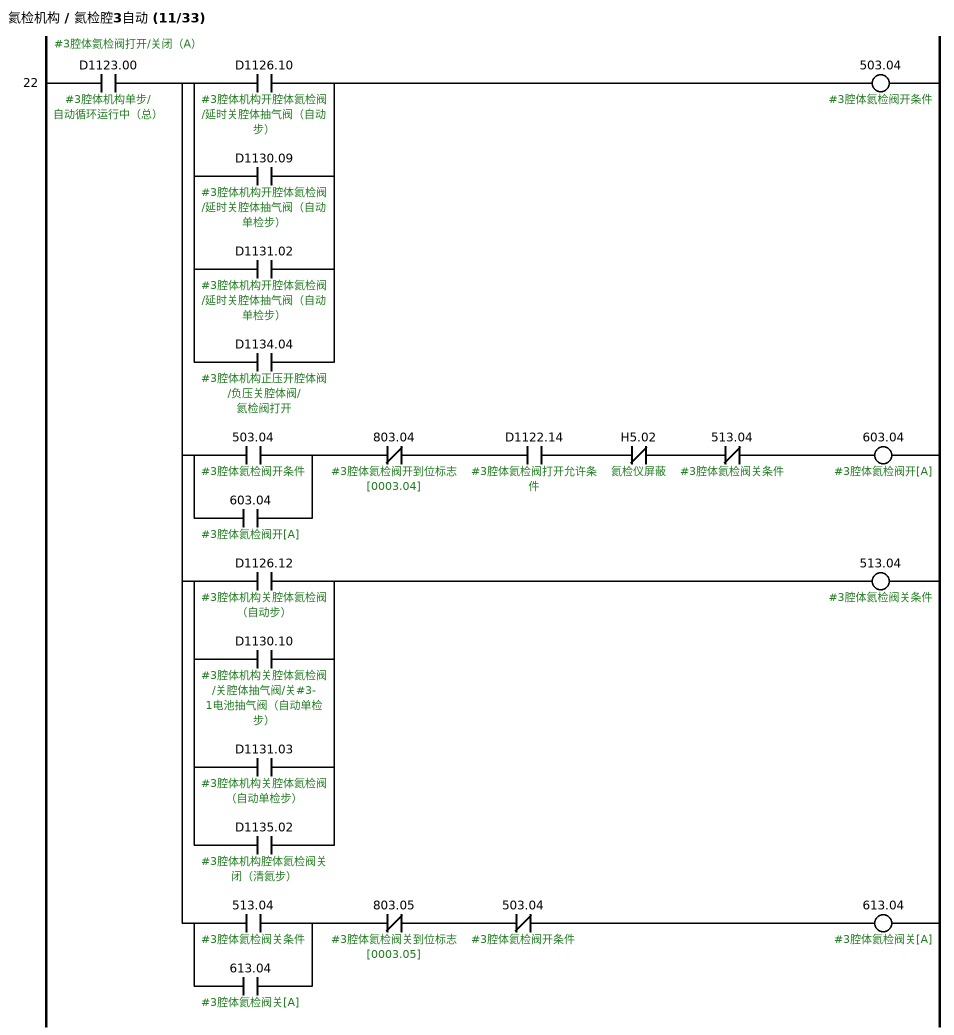
; [picture p312: 氦检机构 / 氦检腔3自动, rungs 22-22]
; rung 22: #3腔体氦检阀打开/关闭（A）
LD D1123.00  ; #3腔体机构单步/自动循环运行中（总）
OUT TR0
LD D1126.10  ; #3腔体机构开腔体氦检阀/延时关腔体抽气阀（自动步）
OR D1130.09  ; #3腔体机构开腔体氦检阀/延时关腔体抽气阀（自动单检步）
OR D1131.02  ; #3腔体机构开腔体氦检阀/延时关腔体抽气阀（自动单检步）
OR D1134.04  ; #3腔体机构正压开腔体阀/负压关腔体阀/氦检阀打开
ANDLD
OUT 503.04  ; #3腔体氦检阀开条件
LD TR0
LD 503.04  ; #3腔体氦检阀开条件
OR 603.04  ; #3腔体氦检阀开[A]
ANDLD
ANDNOT 803.04  ; #3腔体氦检阀开到位标志[0003.04]
AND D1122.14  ; #3腔体氦检阀打开允许条件
ANDNOT H5.02  ; 氦检仪屏蔽
ANDNOT 513.04  ; #3腔体氦检阀关条件
OUT 603.04  ; #3腔体氦检阀开[A]
LD TR0
LD D1126.12  ; #3腔体机构关腔体氦检阀（自动步）
OR D1130.10  ; #3腔体机构关腔体氦检阀/关腔体抽气阀/关#3-1电池抽气阀（自动单检步）
OR D1131.03  ; #3腔体机构关腔体氦检阀（自动单检步）
OR D1135.02  ; #3腔体机构腔体氦检阀关闭（清氦步）
ANDLD
OUT 513.04  ; #3腔体氦检阀关条件
LD TR0
LD 513.04  ; #3腔体氦检阀关条件
OR 613.04  ; #3腔体氦检阀关[A]
ANDLD
ANDNOT 803.05  ; #3腔体氦检阀关到位标志[0003.05]
ANDNOT 503.04  ; #3腔体氦检阀开条件
OUT 613.04  ; #3腔体氦检阀关[A]

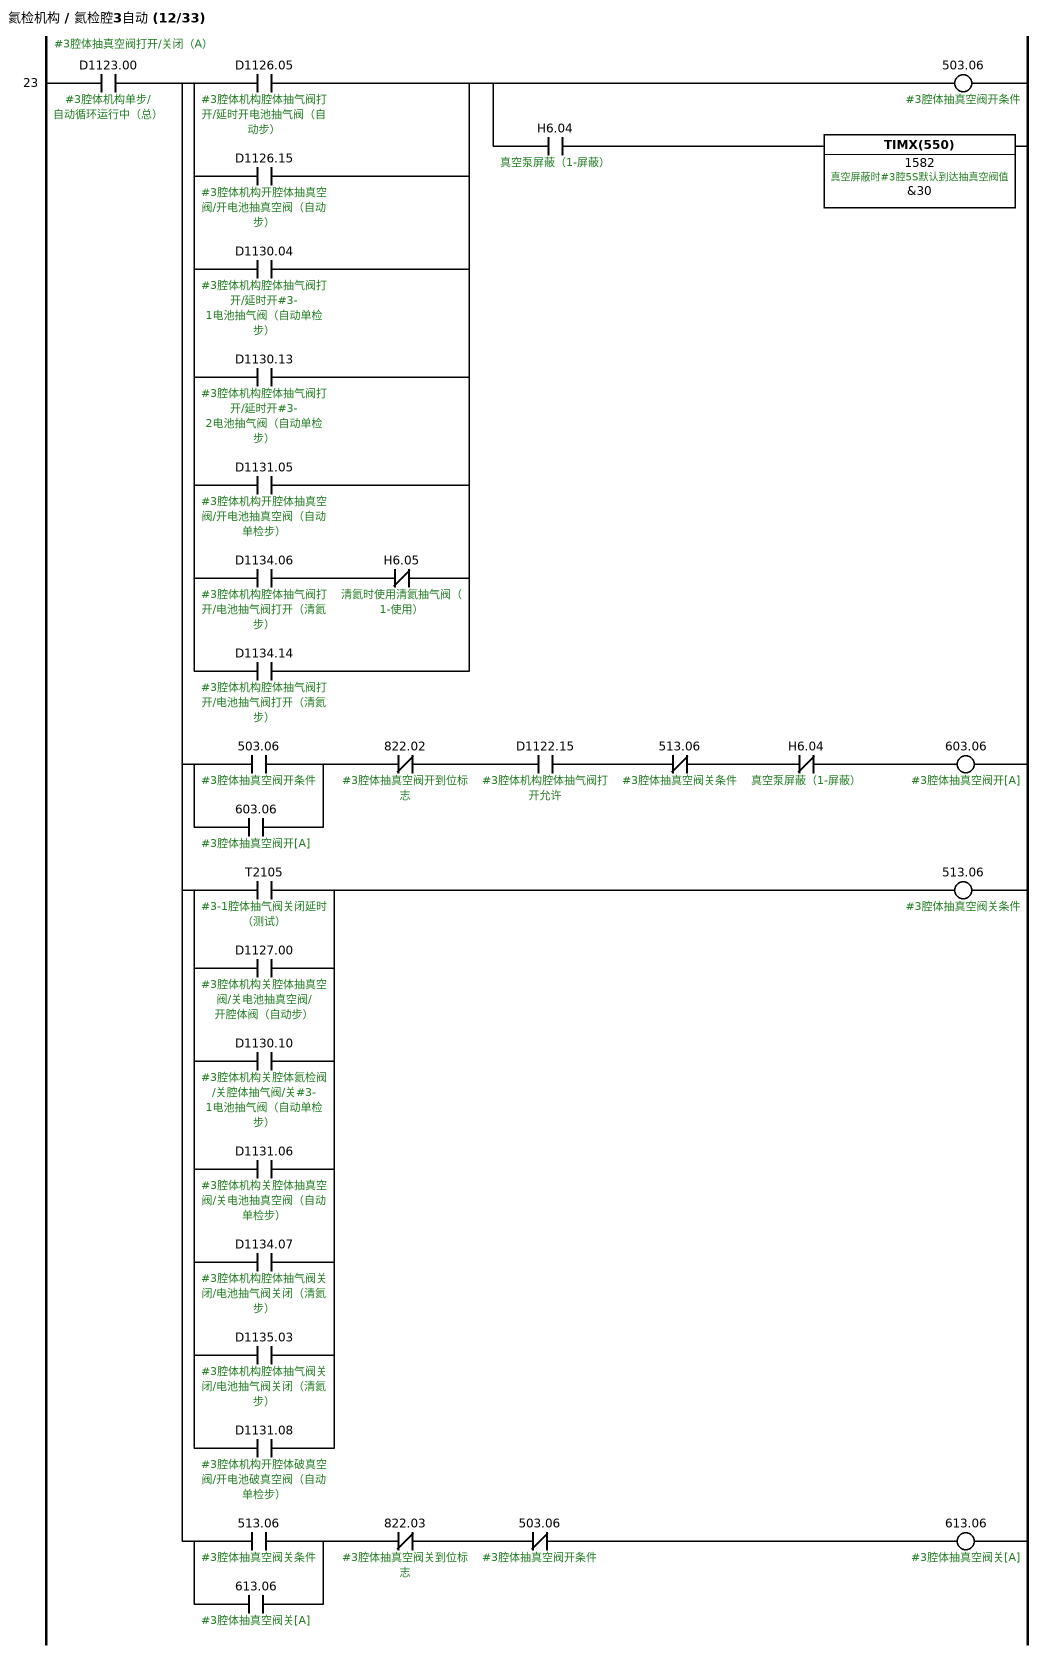
; rung 23: #3腔体抽真空阀打开/关闭（A）
LD D1123.00  ; #3腔体机构单步/自动循环运行中（总）
OUT TR0
LD D1126.05  ; #3腔体机构腔体抽气阀打开/延时开电池抽气阀（自动步）
OR D1126.15  ; #3腔体机构开腔体抽真空阀/开电池抽真空阀（自动步）
OR D1130.04  ; #3腔体机构腔体抽气阀打开/延时开#3-1电池抽气阀（自动单检步）
OR D1130.13  ; #3腔体机构腔体抽气阀打开/延时开#3-2电池抽气阀（自动单检步）
OR D1131.05  ; #3腔体机构开腔体抽真空阀/开电池抽真空阀（自动单检步）
LD D1134.06  ; #3腔体机构腔体抽气阀打开/电池抽气阀打开（清氦步）
ANDNOT H6.05  ; 清氦时使用清氦抽气阀（1-使用）
ORLD
OR D1134.14  ; #3腔体机构腔体抽气阀打开/电池抽气阀打开（清氦步）
ANDLD
OUT 503.06  ; #3腔体抽真空阀开条件
AND H6.04  ; 真空泵屏蔽（1-屏蔽）
TIMX(550) 1582 &30  ; 真空屏蔽时#3腔5S默认到达抽真空阀值
LD TR0
LD 503.06  ; #3腔体抽真空阀开条件
OR 603.06  ; #3腔体抽真空阀开[A]
ANDLD
ANDNOT 822.02  ; #3腔体抽真空阀开到位标志
AND D1122.15  ; #3腔体机构腔体抽气阀打开允许
ANDNOT 513.06  ; #3腔体抽真空阀关条件
ANDNOT H6.04  ; 真空泵屏蔽（1-屏蔽）
OUT 603.06  ; #3腔体抽真空阀开[A]
LD TR0
LD T2105  ; #3-1腔体抽气阀关闭延时（测试）
OR D1127.00  ; #3腔体机构关腔体抽真空阀/关电池抽真空阀/开腔体阀（自动步）
OR D1130.10  ; #3腔体机构关腔体氦检阀/关腔体抽气阀/关#3-1电池抽气阀（自动单检步）
OR D1131.06  ; #3腔体机构关腔体抽真空阀/关电池抽真空阀（自动单检步）
OR D1134.07  ; #3腔体机构腔体抽气阀关闭/电池抽气阀关闭（清氦步）
OR D1135.03  ; #3腔体机构腔体抽气阀关闭/电池抽气阀关闭（清氦步）
OR D1131.08  ; #3腔体机构开腔体破真空阀/开电池破真空阀（自动单检步）
ANDLD
OUT 513.06  ; #3腔体抽真空阀关条件
LD TR0
LD 513.06  ; #3腔体抽真空阀关条件
OR 613.06  ; #3腔体抽真空阀关[A]
ANDLD
ANDNOT 822.03  ; #3腔体抽真空阀关到位标志
ANDNOT 503.06  ; #3腔体抽真空阀开条件
OUT 613.06  ; #3腔体抽真空阀关[A]

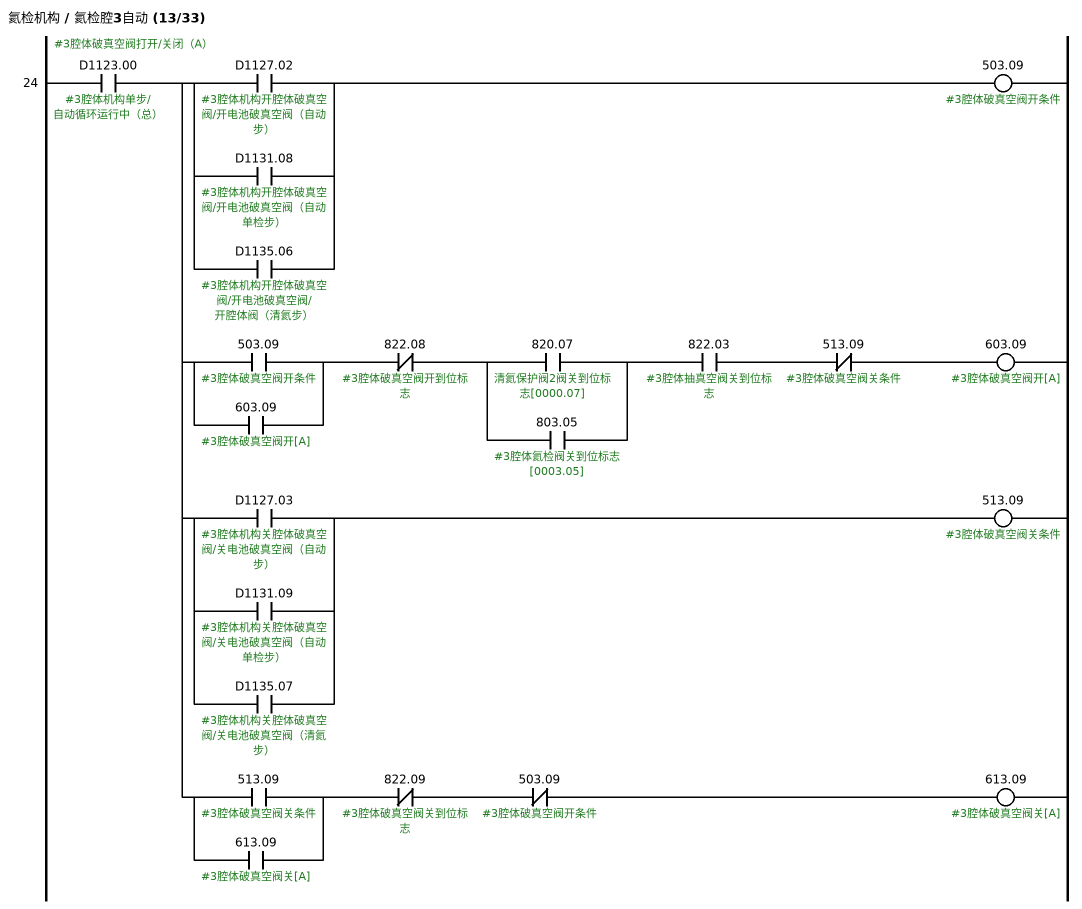
; rung 24: #3腔体破真空阀打开/关闭（A）
LD D1123.00  ; #3腔体机构单步/自动循环运行中（总）
OUT TR0
LD D1127.02  ; #3腔体机构开腔体破真空阀/开电池破真空阀（自动步）
OR D1131.08  ; #3腔体机构开腔体破真空阀/开电池破真空阀（自动单检步）
OR D1135.06  ; #3腔体机构开腔体破真空阀/开电池破真空阀/开腔体阀（清氦步）
ANDLD
OUT 503.09  ; #3腔体破真空阀开条件
LD TR0
LD 503.09  ; #3腔体破真空阀开条件
OR 603.09  ; #3腔体破真空阀开[A]
ANDLD
ANDNOT 822.08  ; #3腔体破真空阀开到位标志
LD 820.07  ; 清氦保护阀2阀关到位标志[0000.07]
OR 803.05  ; #3腔体氦检阀关到位标志[0003.05]
ANDLD
AND 822.03  ; #3腔体抽真空阀关到位标志
ANDNOT 513.09  ; #3腔体破真空阀关条件
OUT 603.09  ; #3腔体破真空阀开[A]
LD TR0
LD D1127.03  ; #3腔体机构关腔体破真空阀/关电池破真空阀（自动步）
OR D1131.09  ; #3腔体机构关腔体破真空阀/关电池破真空阀（自动单检步）
OR D1135.07  ; #3腔体机构关腔体破真空阀/关电池破真空阀（清氦步）
ANDLD
OUT 513.09  ; #3腔体破真空阀关条件
LD TR0
LD 513.09  ; #3腔体破真空阀关条件
OR 613.09  ; #3腔体破真空阀关[A]
ANDLD
ANDNOT 822.09  ; #3腔体破真空阀关到位标志
ANDNOT 503.09  ; #3腔体破真空阀开条件
OUT 613.09  ; #3腔体破真空阀关[A]

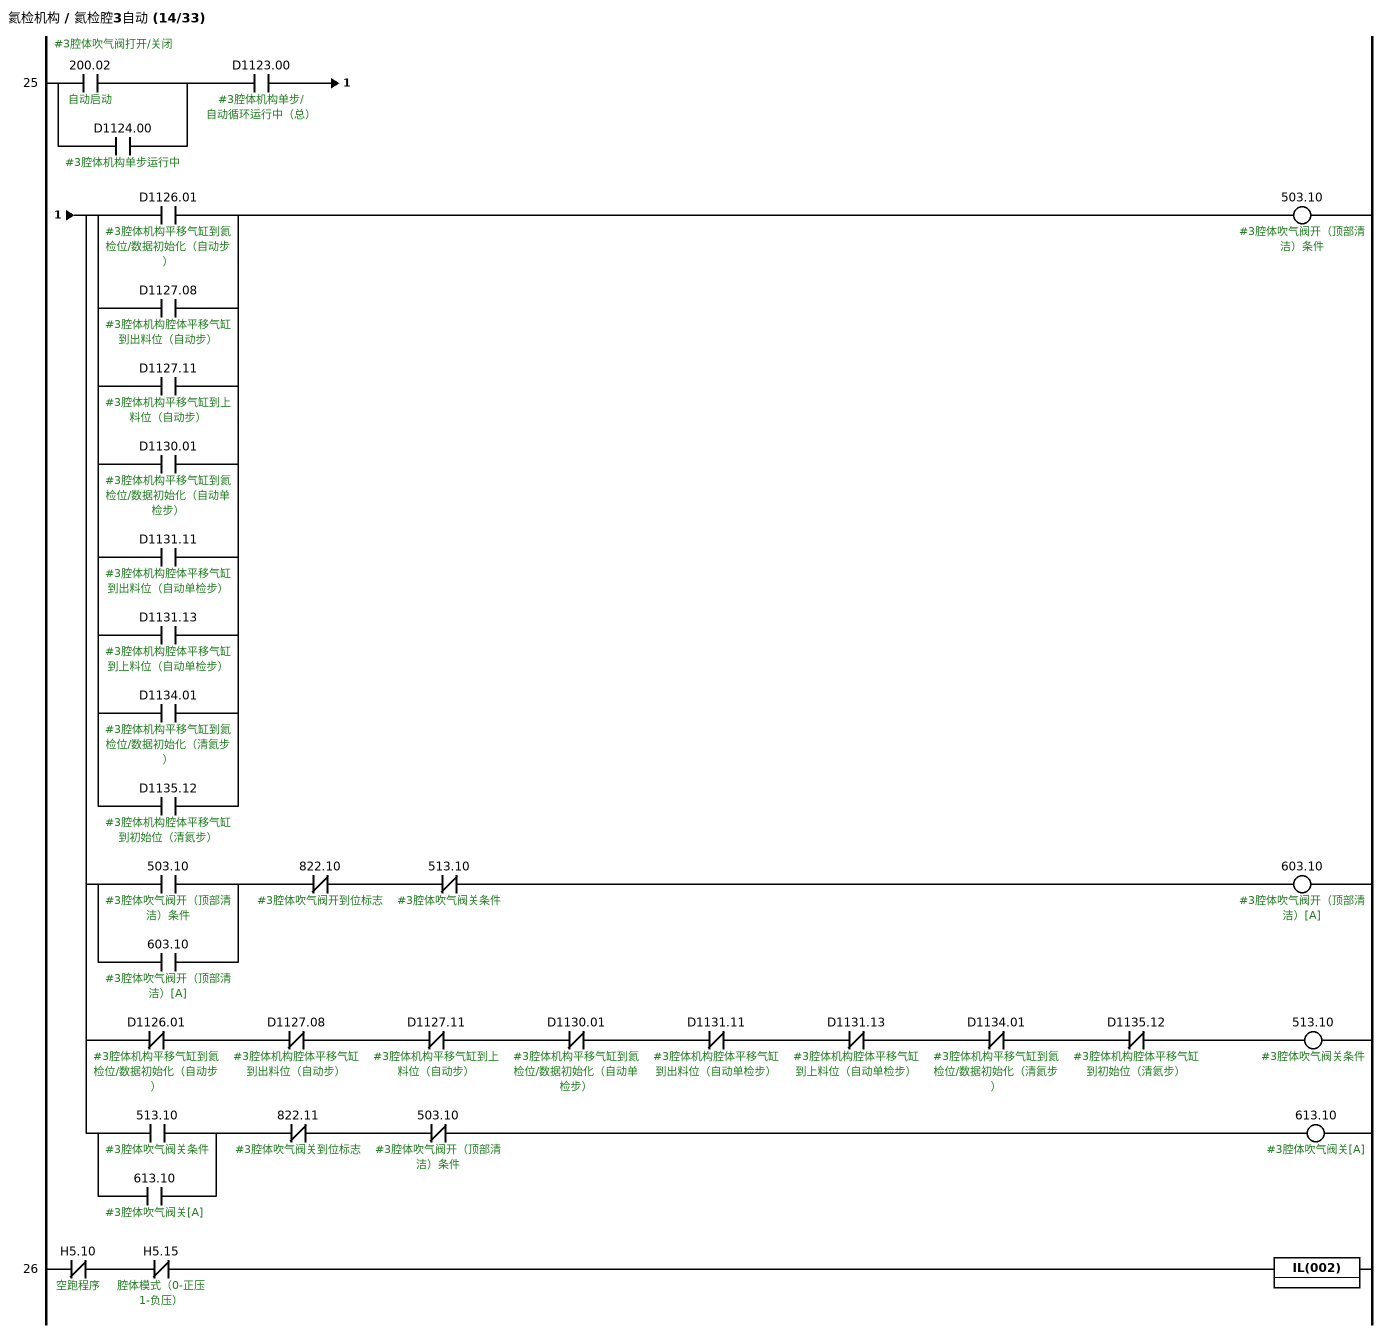
; rung 25: #3腔体吹气阀打开/关闭
LD 200.02  ; 自动启动
OR D1124.00  ; #3腔体机构单步运行中
AND D1123.00  ; #3腔体机构单步/自动循环运行中（总）
OUT TR0
LD D1126.01  ; #3腔体机构平移气缸到氦检位/数据初始化（自动步）
OR D1127.08  ; #3腔体机构腔体平移气缸到出料位（自动步）
OR D1127.11  ; #3腔体机构平移气缸到上料位（自动步）
OR D1130.01  ; #3腔体机构平移气缸到氦检位/数据初始化（自动单检步）
OR D1131.11  ; #3腔体机构腔体平移气缸到出料位（自动单检步）
OR D1131.13  ; #3腔体机构腔体平移气缸到上料位（自动单检步）
OR D1134.01  ; #3腔体机构平移气缸到氦检位/数据初始化（清氦步）
OR D1135.12  ; #3腔体机构腔体平移气缸到初始位（清氦步）
ANDLD
OUT 503.10  ; #3腔体吹气阀开（顶部清洁）条件
LD TR0
LD 503.10  ; #3腔体吹气阀开（顶部清洁）条件
OR 603.10  ; #3腔体吹气阀开（顶部清洁）[A]
ANDLD
ANDNOT 822.10  ; #3腔体吹气阀开到位标志
ANDNOT 513.10  ; #3腔体吹气阀关条件
OUT 603.10  ; #3腔体吹气阀开（顶部清洁）[A]
LD TR0
ANDNOT D1126.01  ; #3腔体机构平移气缸到氦检位/数据初始化（自动步）
ANDNOT D1127.08  ; #3腔体机构腔体平移气缸到出料位（自动步）
ANDNOT D1127.11  ; #3腔体机构平移气缸到上料位（自动步）
ANDNOT D1130.01  ; #3腔体机构平移气缸到氦检位/数据初始化（自动单检步）
ANDNOT D1131.11  ; #3腔体机构腔体平移气缸到出料位（自动单检步）
ANDNOT D1131.13  ; #3腔体机构腔体平移气缸到上料位（自动单检步）
ANDNOT D1134.01  ; #3腔体机构平移气缸到氦检位/数据初始化（清氦步）
ANDNOT D1135.12  ; #3腔体机构腔体平移气缸到初始位（清氦步）
OUT 513.10  ; #3腔体吹气阀关条件
LD TR0
LD 513.10  ; #3腔体吹气阀关条件
OR 613.10  ; #3腔体吹气阀关[A]
ANDLD
ANDNOT 822.11  ; #3腔体吹气阀关到位标志
ANDNOT 503.10  ; #3腔体吹气阀开（顶部清洁）条件
OUT 613.10  ; #3腔体吹气阀关[A]
; rung 26
LDNOT H5.10  ; 空跑程序
ANDNOT H5.15  ; 腔体模式（0-正压 1-负压）
IL(002)

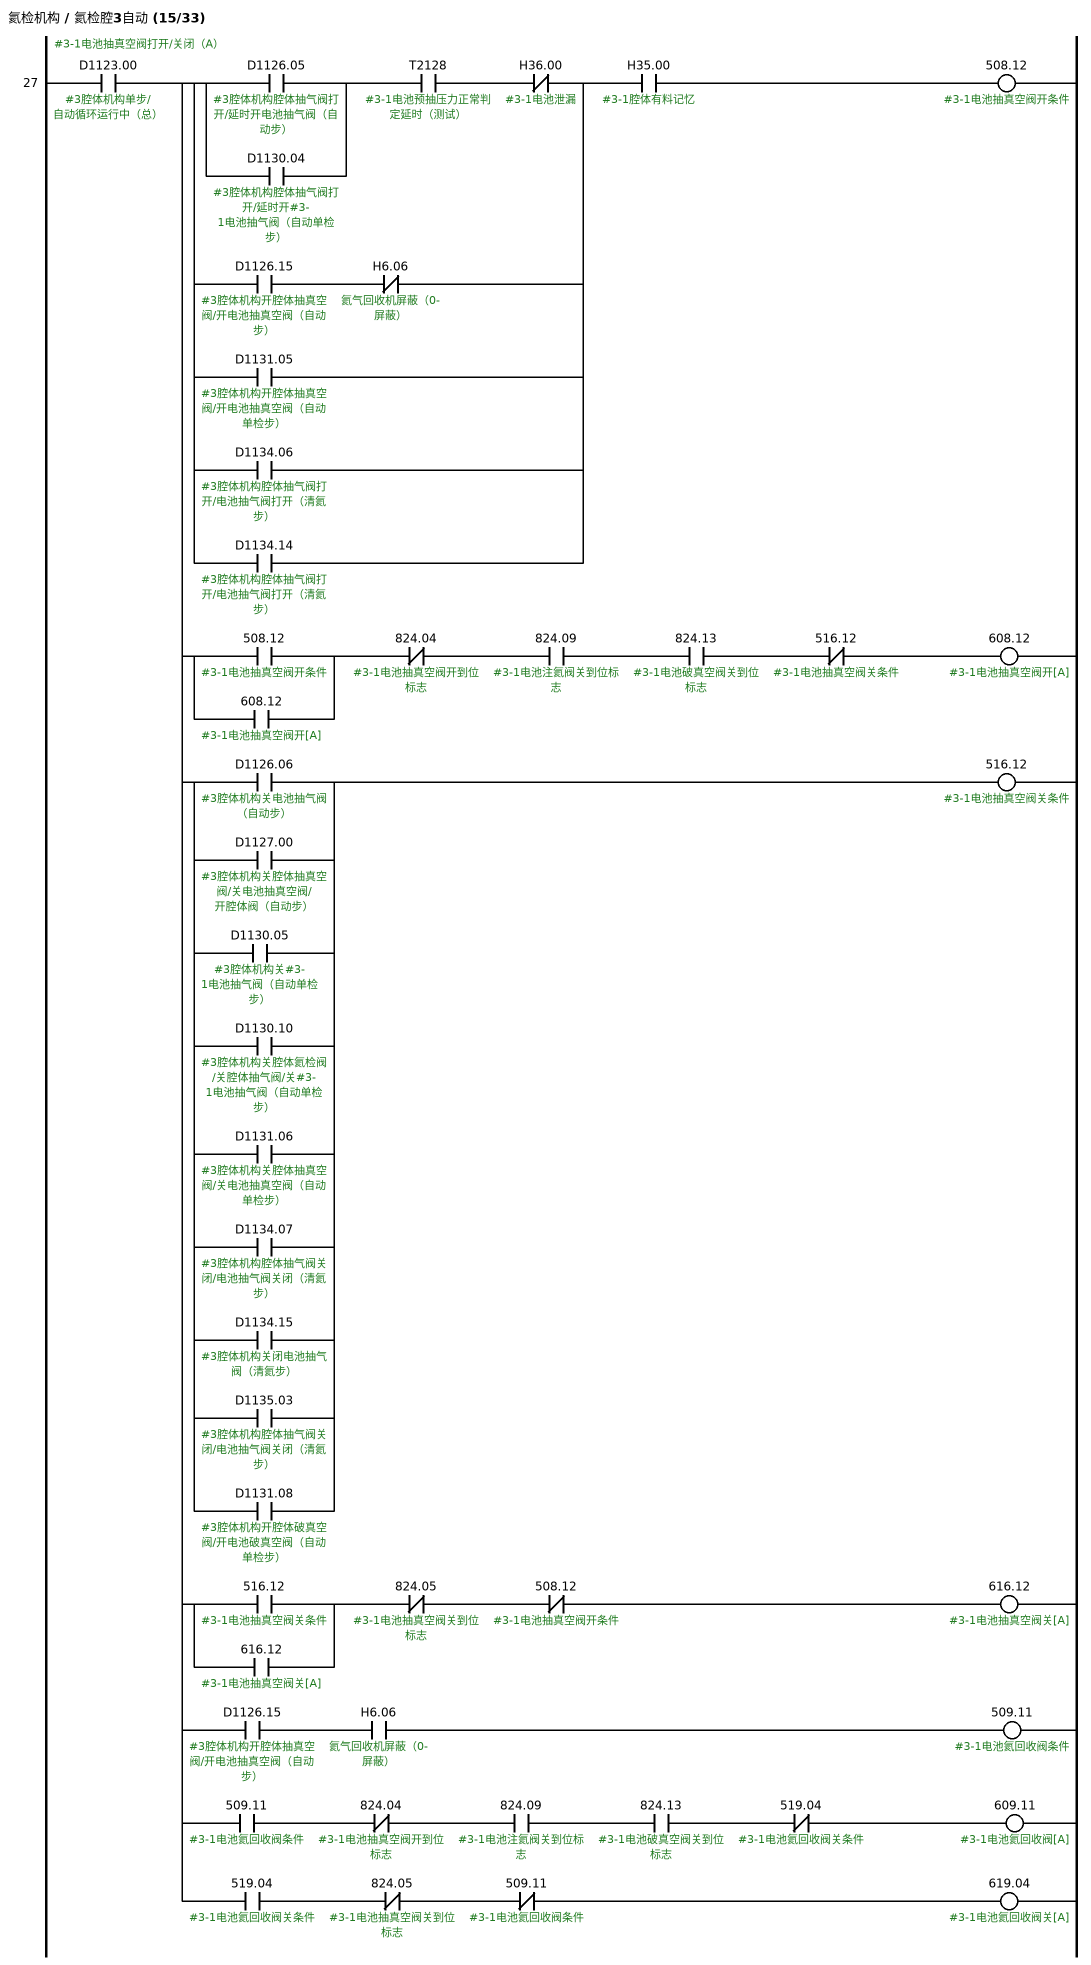
; rung 27: #3-1电池抽真空阀打开/关闭（A）
LD D1123.00  ; #3腔体机构单步/自动循环运行中（总）
OUT TR0
LD D1126.05  ; #3腔体机构腔体抽气阀打开/延时开电池抽气阀（自动步）
OR D1130.04  ; #3腔体机构腔体抽气阀打开/延时开#3-1电池抽气阀（自动单检步）
AND T2128  ; #3-1电池预抽压力正常判定延时（测试）
ANDNOT H36.00  ; #3-1电池泄漏
LD D1126.15  ; #3腔体机构开腔体抽真空阀/开电池抽真空阀（自动步）
ANDNOT H6.06  ; 氦气回收机屏蔽（0-屏蔽）
ORLD
OR D1131.05  ; #3腔体机构开腔体抽真空阀/开电池抽真空阀（自动单检步）
OR D1134.06  ; #3腔体机构腔体抽气阀打开/电池抽气阀打开（清氦步）
OR D1134.14  ; #3腔体机构腔体抽气阀打开/电池抽气阀打开（清氦步）
ANDLD
AND H35.00  ; #3-1腔体有料记忆
OUT 508.12  ; #3-1电池抽真空阀开条件
LD TR0
LD 508.12  ; #3-1电池抽真空阀开条件
OR 608.12  ; #3-1电池抽真空阀开[A]
ANDLD
ANDNOT 824.04  ; #3-1电池抽真空阀开到位标志
AND 824.09  ; #3-1电池注氦阀关到位标志
AND 824.13  ; #3-1电池破真空阀关到位标志
ANDNOT 516.12  ; #3-1电池抽真空阀关条件
OUT 608.12  ; #3-1电池抽真空阀开[A]
LD TR0
LD D1126.06  ; #3腔体机构关电池抽气阀（自动步）
OR D1127.00  ; #3腔体机构关腔体抽真空阀/关电池抽真空阀/开腔体阀（自动步）
OR D1130.05  ; #3腔体机构关#3-1电池抽气阀（自动单检步）
OR D1130.10  ; #3腔体机构关腔体氦检阀/关腔体抽气阀/关#3-1电池抽气阀（自动单检步）
OR D1131.06  ; #3腔体机构关腔体抽真空阀/关电池抽真空阀（自动单检步）
OR D1134.07  ; #3腔体机构腔体抽气阀关闭/电池抽气阀关闭（清氦步）
OR D1134.15  ; #3腔体机构关闭电池抽气阀（清氦步）
OR D1135.03  ; #3腔体机构腔体抽气阀关闭/电池抽气阀关闭（清氦步）
OR D1131.08  ; #3腔体机构开腔体破真空阀/开电池破真空阀（自动单检步）
ANDLD
OUT 516.12  ; #3-1电池抽真空阀关条件
LD TR0
LD 516.12  ; #3-1电池抽真空阀关条件
OR 616.12  ; #3-1电池抽真空阀关[A]
ANDLD
ANDNOT 824.05  ; #3-1电池抽真空阀关到位标志
ANDNOT 508.12  ; #3-1电池抽真空阀开条件
OUT 616.12  ; #3-1电池抽真空阀关[A]
LD TR0
AND D1126.15  ; #3腔体机构开腔体抽真空阀/开电池抽真空阀（自动步）
AND H6.06  ; 氦气回收机屏蔽（0-屏蔽）
OUT 509.11  ; #3-1电池氦回收阀条件
LD TR0
AND 509.11  ; #3-1电池氦回收阀条件
ANDNOT 824.04  ; #3-1电池抽真空阀开到位标志
AND 824.09  ; #3-1电池注氦阀关到位标志
AND 824.13  ; #3-1电池破真空阀关到位标志
ANDNOT 519.04  ; #3-1电池氦回收阀关条件
OUT 609.11  ; #3-1电池氦回收阀[A]
LD TR0
AND 519.04  ; #3-1电池氦回收阀关条件
ANDNOT 824.05  ; #3-1电池抽真空阀关到位标志
ANDNOT 509.11  ; #3-1电池氦回收阀条件
OUT 619.04  ; #3-1电池氦回收阀关[A]

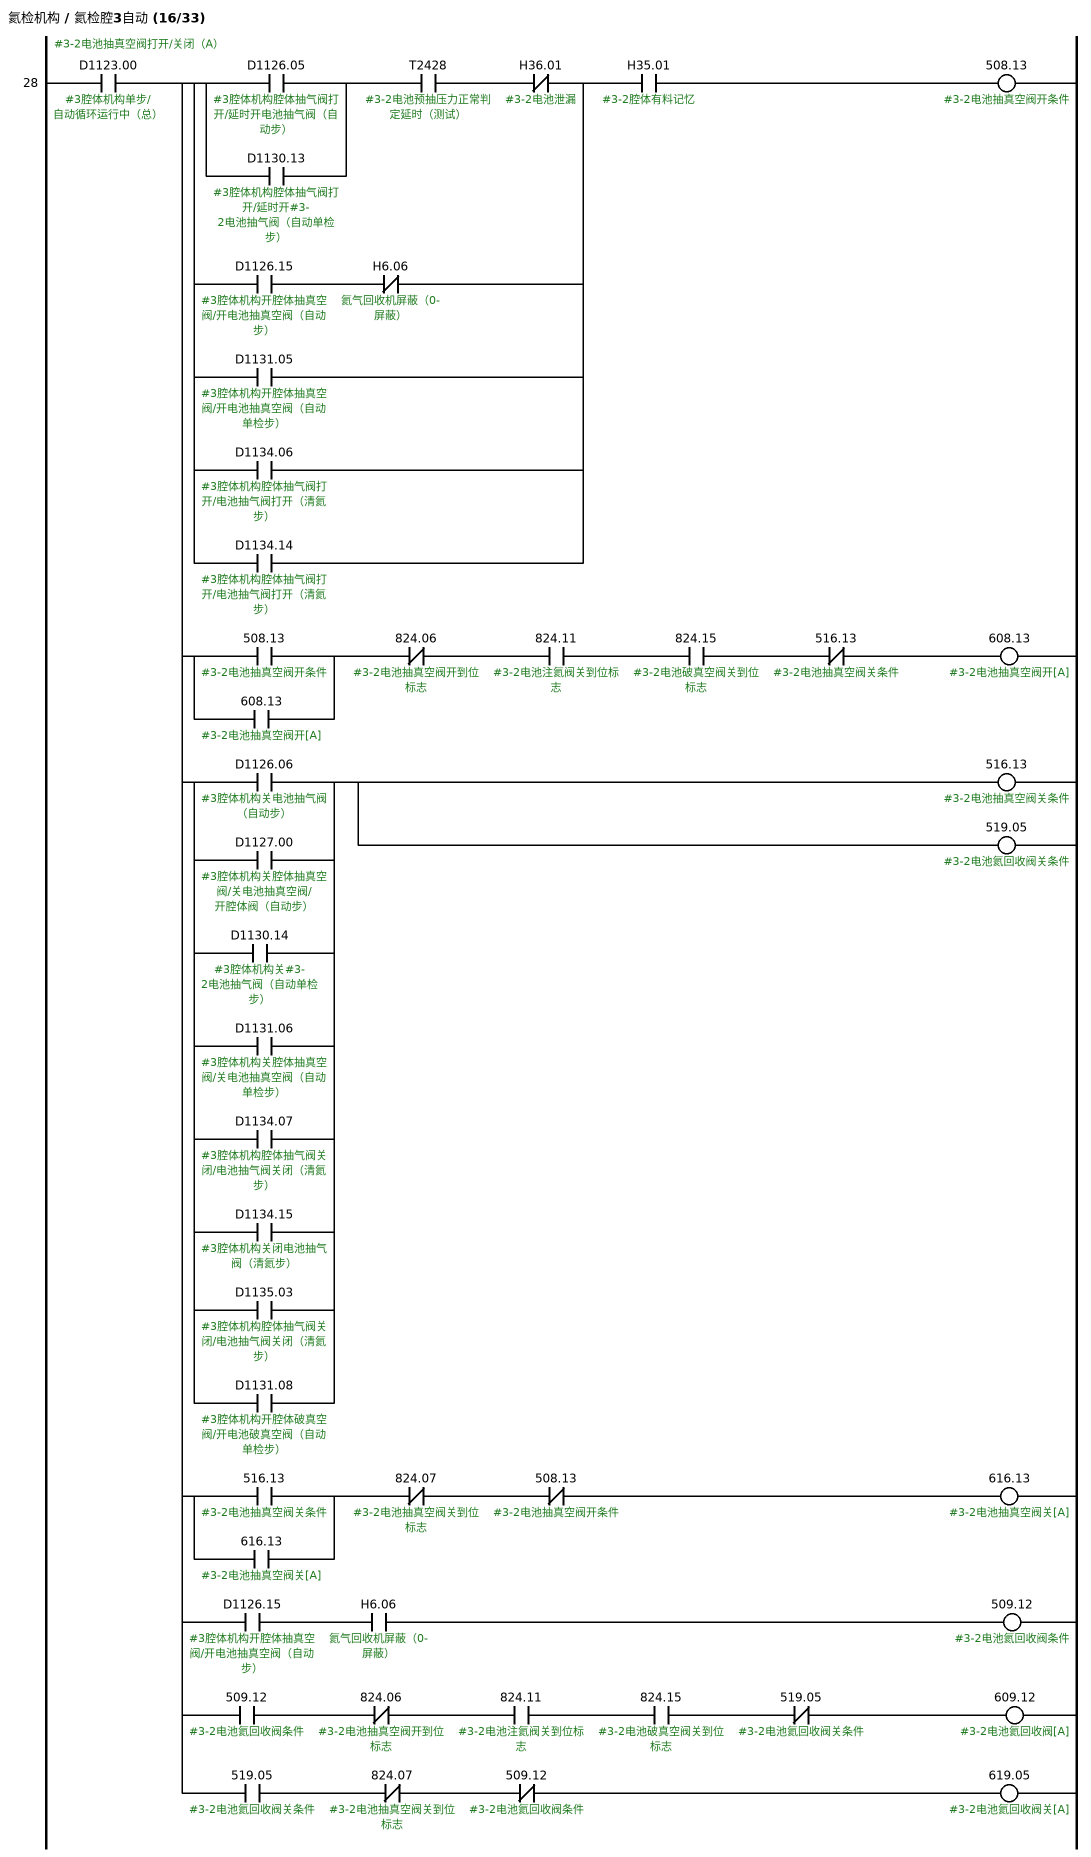
; rung 28: #3-2电池抽真空阀打开/关闭（A）
LD D1123.00  ; #3腔体机构单步/自动循环运行中（总）
OUT TR0
LD D1126.05  ; #3腔体机构腔体抽气阀打开/延时开电池抽气阀（自动步）
OR D1130.13  ; #3腔体机构腔体抽气阀打开/延时开#3-2电池抽气阀（自动单检步）
AND T2428  ; #3-2电池预抽压力正常判定延时（测试）
ANDNOT H36.01  ; #3-2电池泄漏
LD D1126.15  ; #3腔体机构开腔体抽真空阀/开电池抽真空阀（自动步）
ANDNOT H6.06  ; 氦气回收机屏蔽（0-屏蔽）
ORLD
OR D1131.05  ; #3腔体机构开腔体抽真空阀/开电池抽真空阀（自动单检步）
OR D1134.06  ; #3腔体机构腔体抽气阀打开/电池抽气阀打开（清氦步）
OR D1134.14  ; #3腔体机构腔体抽气阀打开/电池抽气阀打开（清氦步）
ANDLD
AND H35.01  ; #3-2腔体有料记忆
OUT 508.13  ; #3-2电池抽真空阀开条件
LD TR0
LD 508.13  ; #3-2电池抽真空阀开条件
OR 608.13  ; #3-2电池抽真空阀开[A]
ANDLD
ANDNOT 824.06  ; #3-2电池抽真空阀开到位标志
AND 824.11  ; #3-2电池注氦阀关到位标志
AND 824.15  ; #3-2电池破真空阀关到位标志
ANDNOT 516.13  ; #3-2电池抽真空阀关条件
OUT 608.13  ; #3-2电池抽真空阀开[A]
LD TR0
LD D1126.06  ; #3腔体机构关电池抽气阀（自动步）
OR D1127.00  ; #3腔体机构关腔体抽真空阀/关电池抽真空阀/开腔体阀（自动步）
OR D1130.14  ; #3腔体机构关#3-2电池抽气阀（自动单检步）
OR D1131.06  ; #3腔体机构关腔体抽真空阀/关电池抽真空阀（自动单检步）
OR D1134.07  ; #3腔体机构腔体抽气阀关闭/电池抽气阀关闭（清氦步）
OR D1134.15  ; #3腔体机构关闭电池抽气阀（清氦步）
OR D1135.03  ; #3腔体机构腔体抽气阀关闭/电池抽气阀关闭（清氦步）
OR D1131.08  ; #3腔体机构开腔体破真空阀/开电池破真空阀（自动单检步）
ANDLD
OUT 516.13  ; #3-2电池抽真空阀关条件
OUT 519.05  ; #3-2电池氦回收阀关条件
LD TR0
LD 516.13  ; #3-2电池抽真空阀关条件
OR 616.13  ; #3-2电池抽真空阀关[A]
ANDLD
ANDNOT 824.07  ; #3-2电池抽真空阀关到位标志
ANDNOT 508.13  ; #3-2电池抽真空阀开条件
OUT 616.13  ; #3-2电池抽真空阀关[A]
LD TR0
AND D1126.15  ; #3腔体机构开腔体抽真空阀/开电池抽真空阀（自动步）
AND H6.06  ; 氦气回收机屏蔽（0-屏蔽）
OUT 509.12  ; #3-2电池氦回收阀条件
LD TR0
AND 509.12  ; #3-2电池氦回收阀条件
ANDNOT 824.06  ; #3-2电池抽真空阀开到位标志
AND 824.11  ; #3-2电池注氦阀关到位标志
AND 824.15  ; #3-2电池破真空阀关到位标志
ANDNOT 519.05  ; #3-2电池氦回收阀关条件
OUT 609.12  ; #3-2电池氦回收阀[A]
LD TR0
AND 519.05  ; #3-2电池氦回收阀关条件
ANDNOT 824.07  ; #3-2电池抽真空阀关到位标志
ANDNOT 509.12  ; #3-2电池氦回收阀条件
OUT 619.05  ; #3-2电池氦回收阀关[A]

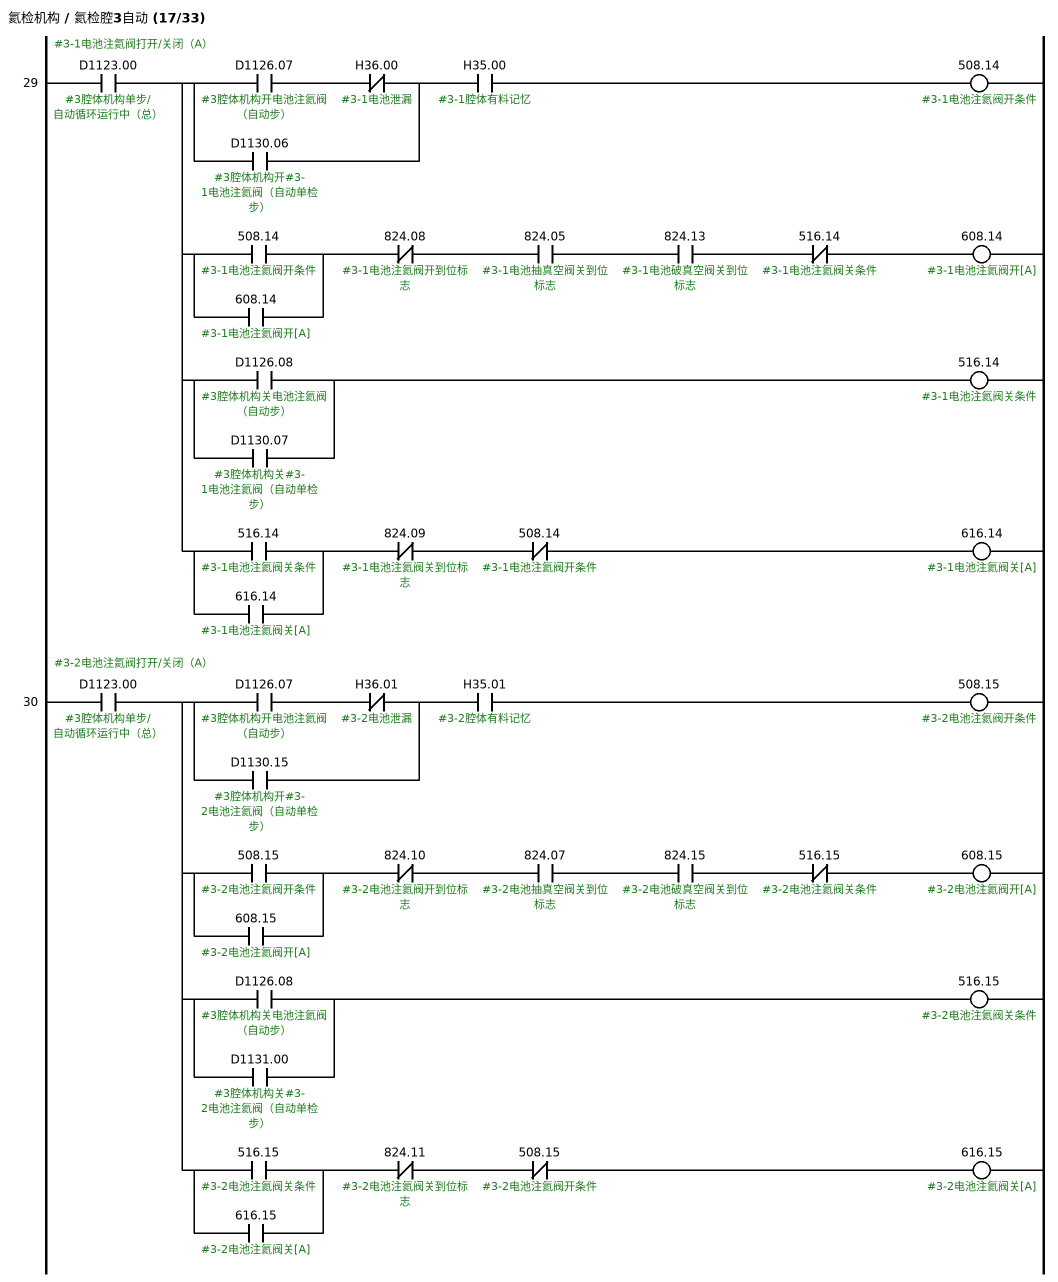
; rung 29: #3-1电池注氦阀打开/关闭（A）
LD D1123.00  ; #3腔体机构单步/自动循环运行中（总）
OUT TR0
LD D1126.07  ; #3腔体机构开电池注氦阀（自动步）
ANDNOT H36.00  ; #3-1电池泄漏
OR D1130.06  ; #3腔体机构开#3-1电池注氦阀（自动单检步）
ANDLD
AND H35.00  ; #3-1腔体有料记忆
OUT 508.14  ; #3-1电池注氦阀开条件
LD TR0
LD 508.14  ; #3-1电池注氦阀开条件
OR 608.14  ; #3-1电池注氦阀开[A]
ANDLD
ANDNOT 824.08  ; #3-1电池注氦阀开到位标志
AND 824.05  ; #3-1电池抽真空阀关到位标志
AND 824.13  ; #3-1电池破真空阀关到位标志
ANDNOT 516.14  ; #3-1电池注氦阀关条件
OUT 608.14  ; #3-1电池注氦阀开[A]
LD TR0
LD D1126.08  ; #3腔体机构关电池注氦阀（自动步）
OR D1130.07  ; #3腔体机构关#3-1电池注氦阀（自动单检步）
ANDLD
OUT 516.14  ; #3-1电池注氦阀关条件
LD TR0
LD 516.14  ; #3-1电池注氦阀关条件
OR 616.14  ; #3-1电池注氦阀关[A]
ANDLD
ANDNOT 824.09  ; #3-1电池注氦阀关到位标志
ANDNOT 508.14  ; #3-1电池注氦阀开条件
OUT 616.14  ; #3-1电池注氦阀关[A]
; rung 30: #3-2电池注氦阀打开/关闭（A）
LD D1123.00  ; #3腔体机构单步/自动循环运行中（总）
OUT TR0
LD D1126.07  ; #3腔体机构开电池注氦阀（自动步）
ANDNOT H36.01  ; #3-2电池泄漏
OR D1130.15  ; #3腔体机构开#3-2电池注氦阀（自动单检步）
ANDLD
AND H35.01  ; #3-2腔体有料记忆
OUT 508.15  ; #3-2电池注氦阀开条件
LD TR0
LD 508.15  ; #3-2电池注氦阀开条件
OR 608.15  ; #3-2电池注氦阀开[A]
ANDLD
ANDNOT 824.10  ; #3-2电池注氦阀开到位标志
AND 824.07  ; #3-2电池抽真空阀关到位标志
AND 824.15  ; #3-2电池破真空阀关到位标志
ANDNOT 516.15  ; #3-2电池注氦阀关条件
OUT 608.15  ; #3-2电池注氦阀开[A]
LD TR0
LD D1126.08  ; #3腔体机构关电池注氦阀（自动步）
OR D1131.00  ; #3腔体机构关#3-2电池注氦阀（自动单检步）
ANDLD
OUT 516.15  ; #3-2电池注氦阀关条件
LD TR0
LD 516.15  ; #3-2电池注氦阀关条件
OR 616.15  ; #3-2电池注氦阀关[A]
ANDLD
ANDNOT 824.11  ; #3-2电池注氦阀关到位标志
ANDNOT 508.15  ; #3-2电池注氦阀开条件
OUT 616.15  ; #3-2电池注氦阀关[A]

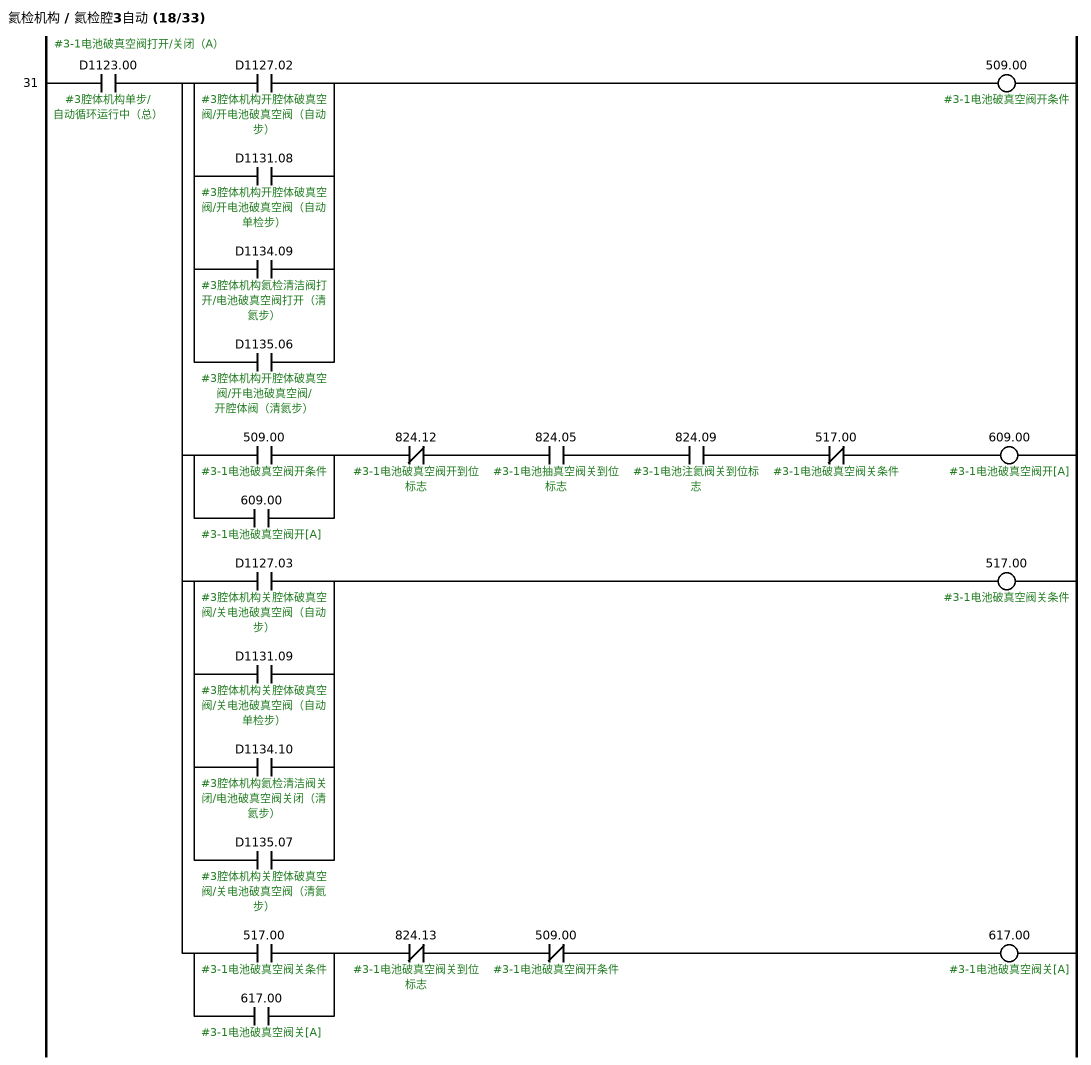
; rung 31: #3-1电池破真空阀打开/关闭（A）
LD D1123.00  ; #3腔体机构单步/自动循环运行中（总）
OUT TR0
LD D1127.02  ; #3腔体机构开腔体破真空阀/开电池破真空阀（自动步）
OR D1131.08  ; #3腔体机构开腔体破真空阀/开电池破真空阀（自动单检步）
OR D1134.09  ; #3腔体机构氦检清洁阀打开/电池破真空阀打开（清氦步）
OR D1135.06  ; #3腔体机构开腔体破真空阀/开电池破真空阀/开腔体阀（清氦步）
ANDLD
OUT 509.00  ; #3-1电池破真空阀开条件
LD TR0
LD 509.00  ; #3-1电池破真空阀开条件
OR 609.00  ; #3-1电池破真空阀开[A]
ANDLD
ANDNOT 824.12  ; #3-1电池破真空阀开到位标志
AND 824.05  ; #3-1电池抽真空阀关到位标志
AND 824.09  ; #3-1电池注氦阀关到位标志
ANDNOT 517.00  ; #3-1电池破真空阀关条件
OUT 609.00  ; #3-1电池破真空阀开[A]
LD TR0
LD D1127.03  ; #3腔体机构关腔体破真空阀/关电池破真空阀（自动步）
OR D1131.09  ; #3腔体机构关腔体破真空阀/关电池破真空阀（自动单检步）
OR D1134.10  ; #3腔体机构氦检清洁阀关闭/电池破真空阀关闭（清氦步）
OR D1135.07  ; #3腔体机构关腔体破真空阀/关电池破真空阀（清氦步）
ANDLD
OUT 517.00  ; #3-1电池破真空阀关条件
LD TR0
LD 517.00  ; #3-1电池破真空阀关条件
OR 617.00  ; #3-1电池破真空阀关[A]
ANDLD
ANDNOT 824.13  ; #3-1电池破真空阀关到位标志
ANDNOT 509.00  ; #3-1电池破真空阀开条件
OUT 617.00  ; #3-1电池破真空阀关[A]

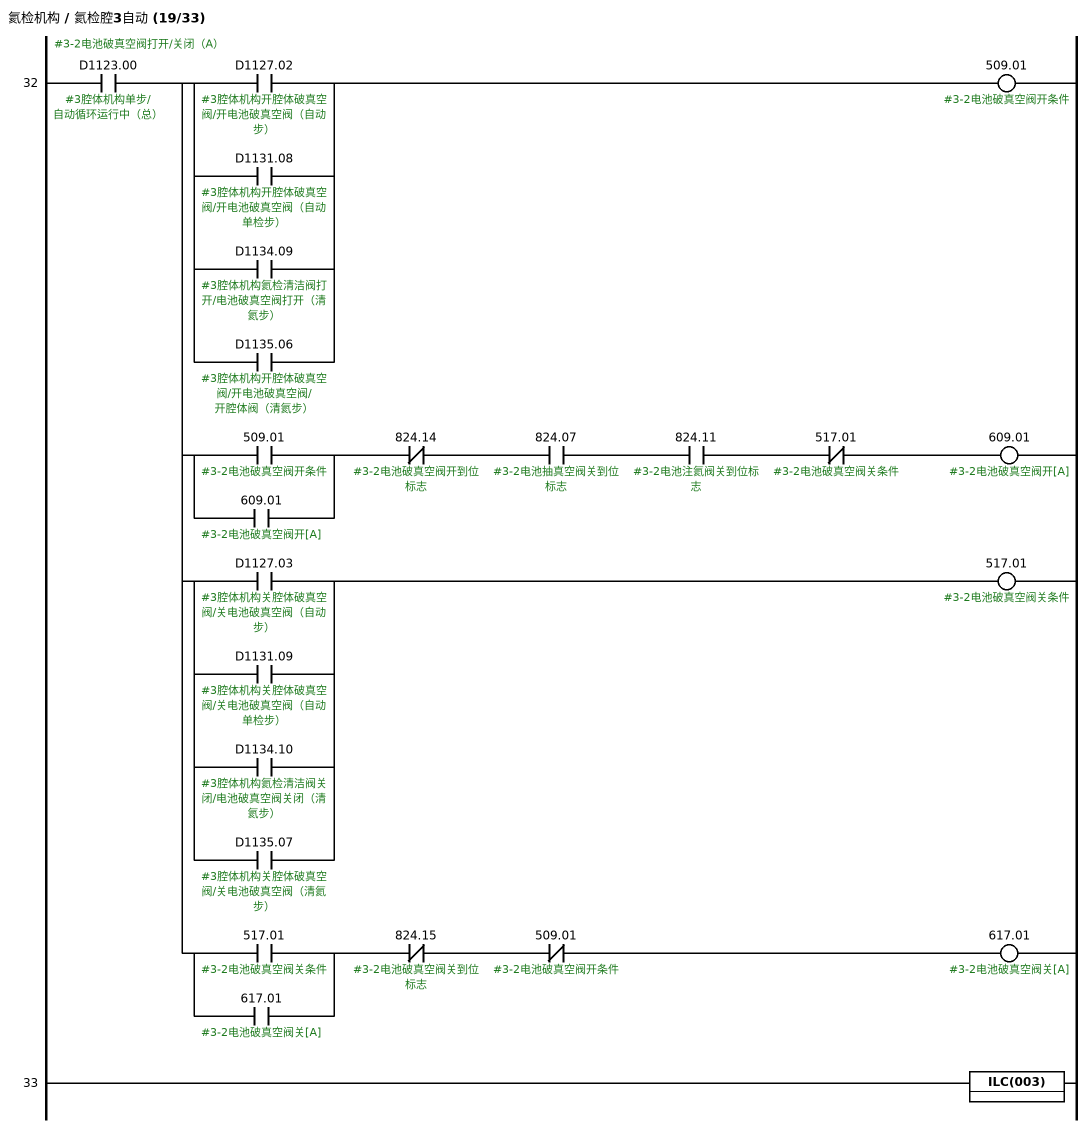
; rung 32: #3-2电池破真空阀打开/关闭（A）
LD D1123.00  ; #3腔体机构单步/自动循环运行中（总）
OUT TR0
LD D1127.02  ; #3腔体机构开腔体破真空阀/开电池破真空阀（自动步）
OR D1131.08  ; #3腔体机构开腔体破真空阀/开电池破真空阀（自动单检步）
OR D1134.09  ; #3腔体机构氦检清洁阀打开/电池破真空阀打开（清氦步）
OR D1135.06  ; #3腔体机构开腔体破真空阀/开电池破真空阀/开腔体阀（清氦步）
ANDLD
OUT 509.01  ; #3-2电池破真空阀开条件
LD TR0
LD 509.01  ; #3-2电池破真空阀开条件
OR 609.01  ; #3-2电池破真空阀开[A]
ANDLD
ANDNOT 824.14  ; #3-2电池破真空阀开到位标志
AND 824.07  ; #3-2电池抽真空阀关到位标志
AND 824.11  ; #3-2电池注氦阀关到位标志
ANDNOT 517.01  ; #3-2电池破真空阀关条件
OUT 609.01  ; #3-2电池破真空阀开[A]
LD TR0
LD D1127.03  ; #3腔体机构关腔体破真空阀/关电池破真空阀（自动步）
OR D1131.09  ; #3腔体机构关腔体破真空阀/关电池破真空阀（自动单检步）
OR D1134.10  ; #3腔体机构氦检清洁阀关闭/电池破真空阀关闭（清氦步）
OR D1135.07  ; #3腔体机构关腔体破真空阀/关电池破真空阀（清氦步）
ANDLD
OUT 517.01  ; #3-2电池破真空阀关条件
LD TR0
LD 517.01  ; #3-2电池破真空阀关条件
OR 617.01  ; #3-2电池破真空阀关[A]
ANDLD
ANDNOT 824.15  ; #3-2电池破真空阀关到位标志
ANDNOT 509.01  ; #3-2电池破真空阀开条件
OUT 617.01  ; #3-2电池破真空阀关[A]
; rung 33
ILC(003)

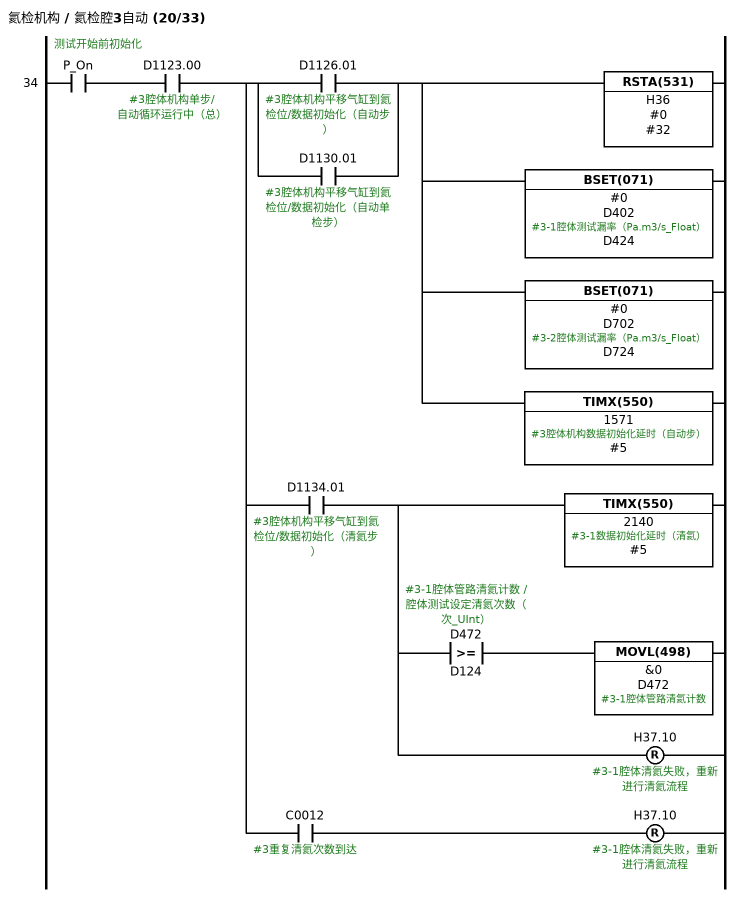
; rung 34: 测试开始前初始化
LD P_On
AND D1123.00  ; #3腔体机构单步/自动循环运行中（总）
OUT TR0
LD D1126.01  ; #3腔体机构平移气缸到氦检位/数据初始化（自动步）
OR D1130.01  ; #3腔体机构平移气缸到氦检位/数据初始化（自动单检步）
ANDLD
RSTA(531) H36 #0 #32
BSET(071) #0 D402 D424  ; #3-1腔体测试漏率（Pa.m3/s_Float）
BSET(071) #0 D702 D724  ; #3-2腔体测试漏率（Pa.m3/s_Float）
TIMX(550) 1571 #5  ; #3腔体机构数据初始化延时（自动步）
LD TR0
AND D1134.01  ; #3腔体机构平移气缸到氦检位/数据初始化（清氦步）
OUT TR1
TIMX(550) 2140 #5  ; #3-1数据初始化延时（清氦）
AND>=(325) D472 D124  ; #3-1腔体管路清氦计数, 腔体测试设定清氦次数（次_UInt）
MOVL(498) &0 D472  ; #3-1腔体管路清氦计数
LD TR1
RSET H37.10  ; #3-1腔体清氦失败，重新进行清氦流程
LD TR0
AND C0012  ; #3重复清氦次数到达
RSET H37.10  ; #3-1腔体清氦失败，重新进行清氦流程

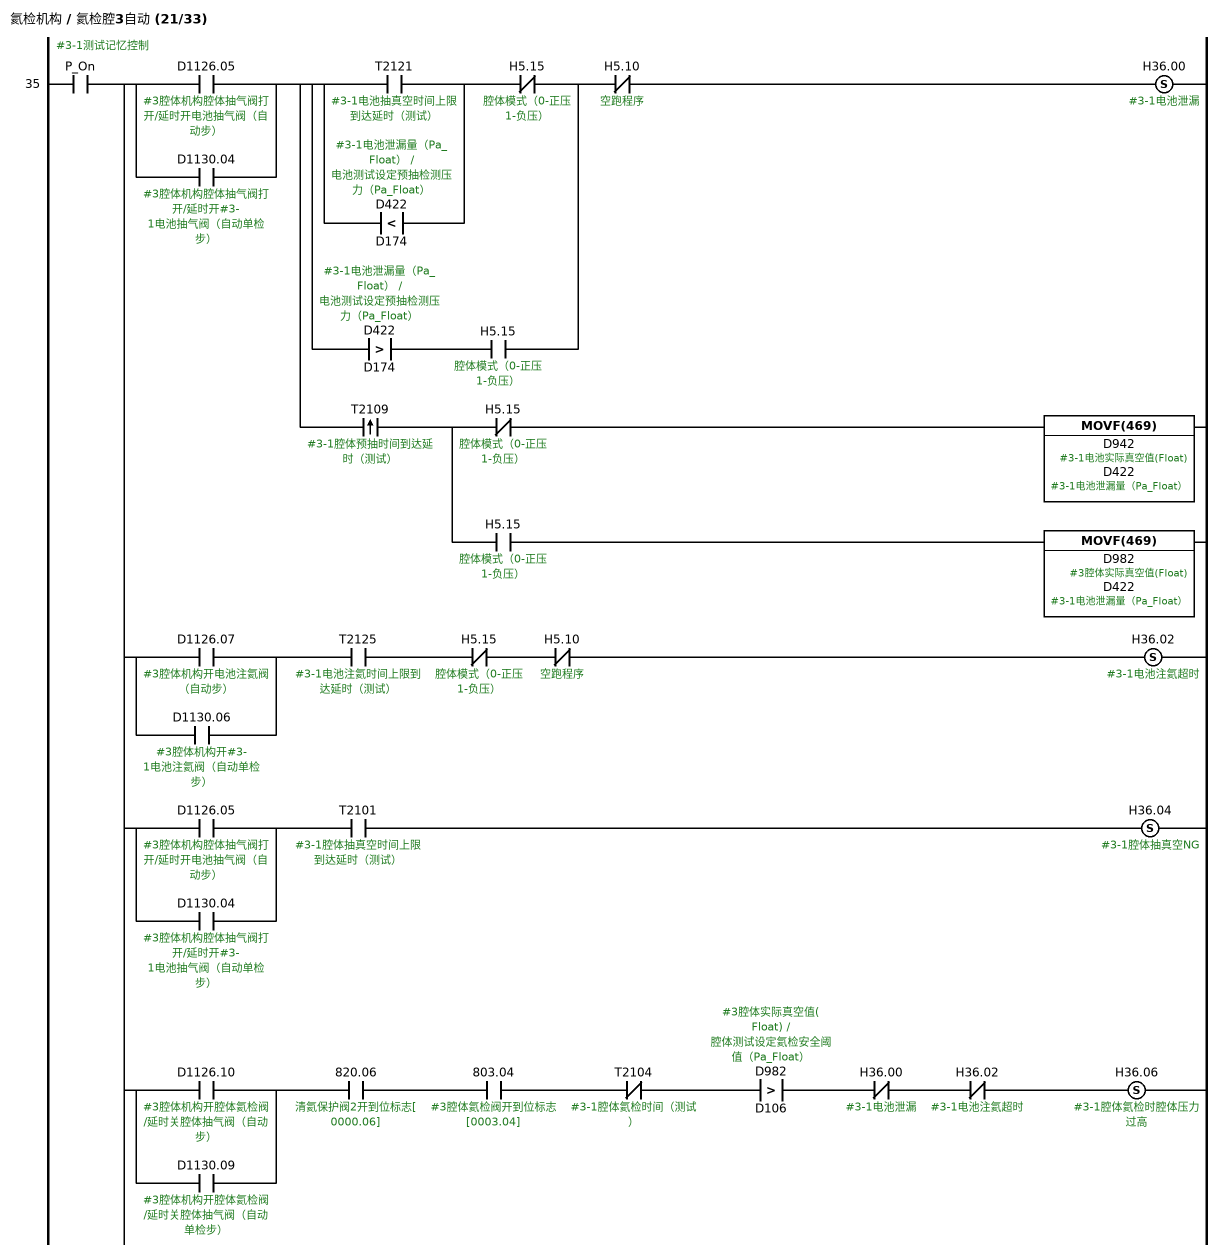

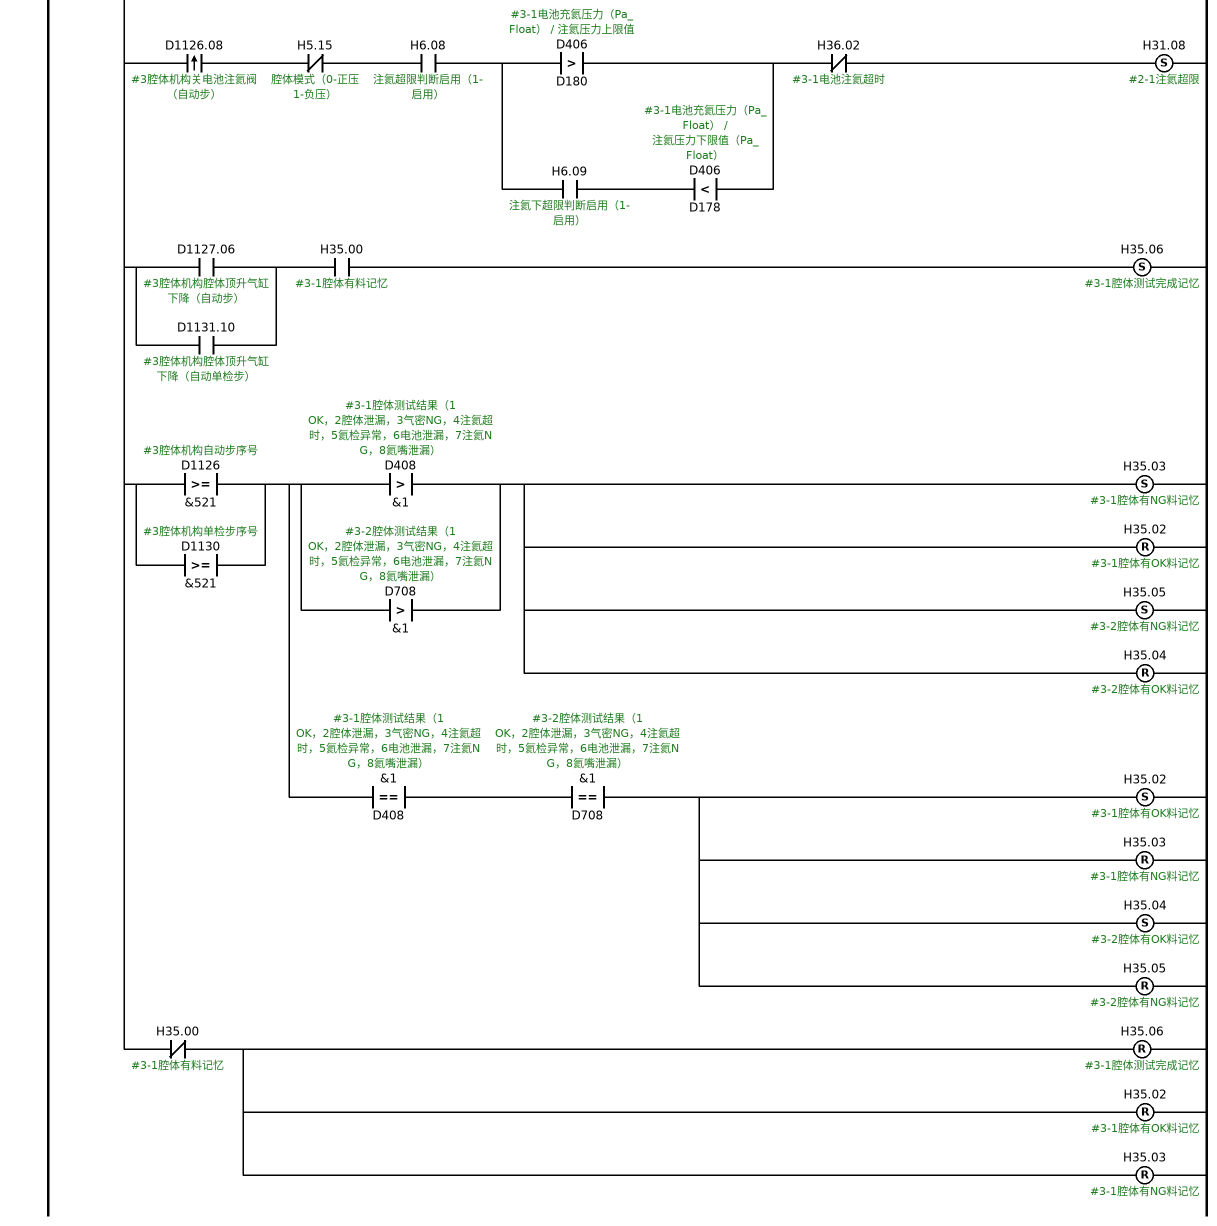
; rung 35: #3-1测试记忆控制
LD P_On
OUT TR0
LD D1126.05  ; #3腔体机构腔体抽气阀打开/延时开电池抽气阀（自动步）
OR D1130.04  ; #3腔体机构腔体抽气阀打开/延时开#3-1电池抽气阀（自动单检步）
ANDLD
OUT TR1
LD T2121  ; #3-1电池抽真空时间上限到达延时（测试）
OR<F(331) D422 D174  ; #3-1电池泄漏量（Pa_Float）, 电池测试设定预抽检测压力（Pa_Float）
ANDNOT H5.15  ; 腔体模式（0-正压 1-负压）
LD>F(333) D422 D174  ; #3-1电池泄漏量（Pa_Float）, 电池测试设定预抽检测压力（Pa_Float）
AND H5.15  ; 腔体模式（0-正压 1-负压）
ORLD
ANDLD
ANDNOT H5.10  ; 空跑程序
SET H36.00  ; #3-1电池泄漏
LD TR1
@AND T2109  ; #3-1腔体预抽时间到达延时（测试）
OUT TR1
ANDNOT H5.15  ; 腔体模式（0-正压 1-负压）
MOVF(469) D942 D422  ; #3-1电池实际真空值(Float), #3-1电池泄漏量（Pa_Float）
LD TR1
AND H5.15  ; 腔体模式（0-正压 1-负压）
MOVF(469) D982 D422  ; #3腔体实际真空值(Float), #3-1电池泄漏量（Pa_Float）
LD TR0
LD D1126.07  ; #3腔体机构开电池注氦阀（自动步）
OR D1130.06  ; #3腔体机构开#3-1电池注氦阀（自动单检步）
ANDLD
AND T2125  ; #3-1电池注氦时间上限到达延时（测试）
ANDNOT H5.15  ; 腔体模式（0-正压 1-负压）
ANDNOT H5.10  ; 空跑程序
SET H36.02  ; #3-1电池注氦超时
LD TR0
LD D1126.05  ; #3腔体机构腔体抽气阀打开/延时开电池抽气阀（自动步）
OR D1130.04  ; #3腔体机构腔体抽气阀打开/延时开#3-1电池抽气阀（自动单检步）
ANDLD
AND T2101  ; #3-1腔体抽真空时间上限到达延时（测试）
SET H36.04  ; #3-1腔体抽真空NG
LD TR0
LD D1126.10  ; #3腔体机构开腔体氦检阀/延时关腔体抽气阀（自动步）
OR D1130.09  ; #3腔体机构开腔体氦检阀/延时关腔体抽气阀（自动单检步）
ANDLD
AND 820.06  ; 清氦保护阀2开到位标志[0000.06]
AND 803.04  ; #3腔体氦检阀开到位标志[0003.04]
ANDNOT T2104  ; #3-1腔体氦检时间（测试）
AND>F(333) D982 D106  ; #3腔体实际真空值(Float), 腔体测试设定氦检安全阈值（Pa_Float）
ANDNOT H36.00  ; #3-1电池泄漏
ANDNOT H36.02  ; #3-1电池注氦超时
SET H36.06  ; #3-1腔体氦检时腔体压力过高
LD TR0
@AND D1126.08  ; #3腔体机构关电池注氦阀（自动步）
ANDNOT H5.15  ; 腔体模式（0-正压 1-负压）
AND H6.08  ; 注氦超限判断启用（1-启用）
LD>F(333) D406 D180  ; #3-1电池充氦压力（Pa_Float）, 注氦压力上限值
LD H6.09  ; 注氦下超限判断启用（1-启用）
AND<F(331) D406 D178  ; #3-1电池充氦压力（Pa_Float）, 注氦压力下限值（Pa_Float）
ORLD
ANDLD
ANDNOT H36.02  ; #3-1电池注氦超时
SET H31.08  ; #2-1注氦超限
LD TR0
LD D1127.06  ; #3腔体机构腔体顶升气缸下降（自动步）
OR D1131.10  ; #3腔体机构腔体顶升气缸下降（自动单检步）
ANDLD
AND H35.00  ; #3-1腔体有料记忆
SET H35.06  ; #3-1腔体测试完成记忆
LD TR0
LD>=L(326) D1126 &521  ; #3腔体机构自动步序号
OR>=L(326) D1130 &521  ; #3腔体机构单检步序号
ANDLD
OUT TR1
LD>(320) D408 &1  ; #3-1腔体测试结果（1 OK，2腔体泄漏，3气密NG，4注氦超时，5氦检异常，6电池泄漏，7注氦NG，8氦嘴泄漏）
OR>(320) D708 &1  ; #3-2腔体测试结果（1 OK，2腔体泄漏，3气密NG，4注氦超时，5氦检异常，6电池泄漏，7注氦NG，8氦嘴泄漏）
ANDLD
SET H35.03  ; #3-1腔体有NG料记忆
RSET H35.02  ; #3-1腔体有OK料记忆
SET H35.05  ; #3-2腔体有NG料记忆
RSET H35.04  ; #3-2腔体有OK料记忆
LD TR1
AND=(300) &1 D408  ; #3-1腔体测试结果（1 OK，2腔体泄漏，3气密NG，4注氦超时，5氦检异常，6电池泄漏，7注氦NG，8氦嘴泄漏）
AND=(300) &1 D708  ; #3-2腔体测试结果（1 OK，2腔体泄漏，3气密NG，4注氦超时，5氦检异常，6电池泄漏，7注氦NG，8氦嘴泄漏）
SET H35.02  ; #3-1腔体有OK料记忆
RSET H35.03  ; #3-1腔体有NG料记忆
SET H35.04  ; #3-2腔体有OK料记忆
RSET H35.05  ; #3-2腔体有NG料记忆
LD TR0
ANDNOT H35.00  ; #3-1腔体有料记忆
RSET H35.06  ; #3-1腔体测试完成记忆
RSET H35.02  ; #3-1腔体有OK料记忆
RSET H35.03  ; #3-1腔体有NG料记忆

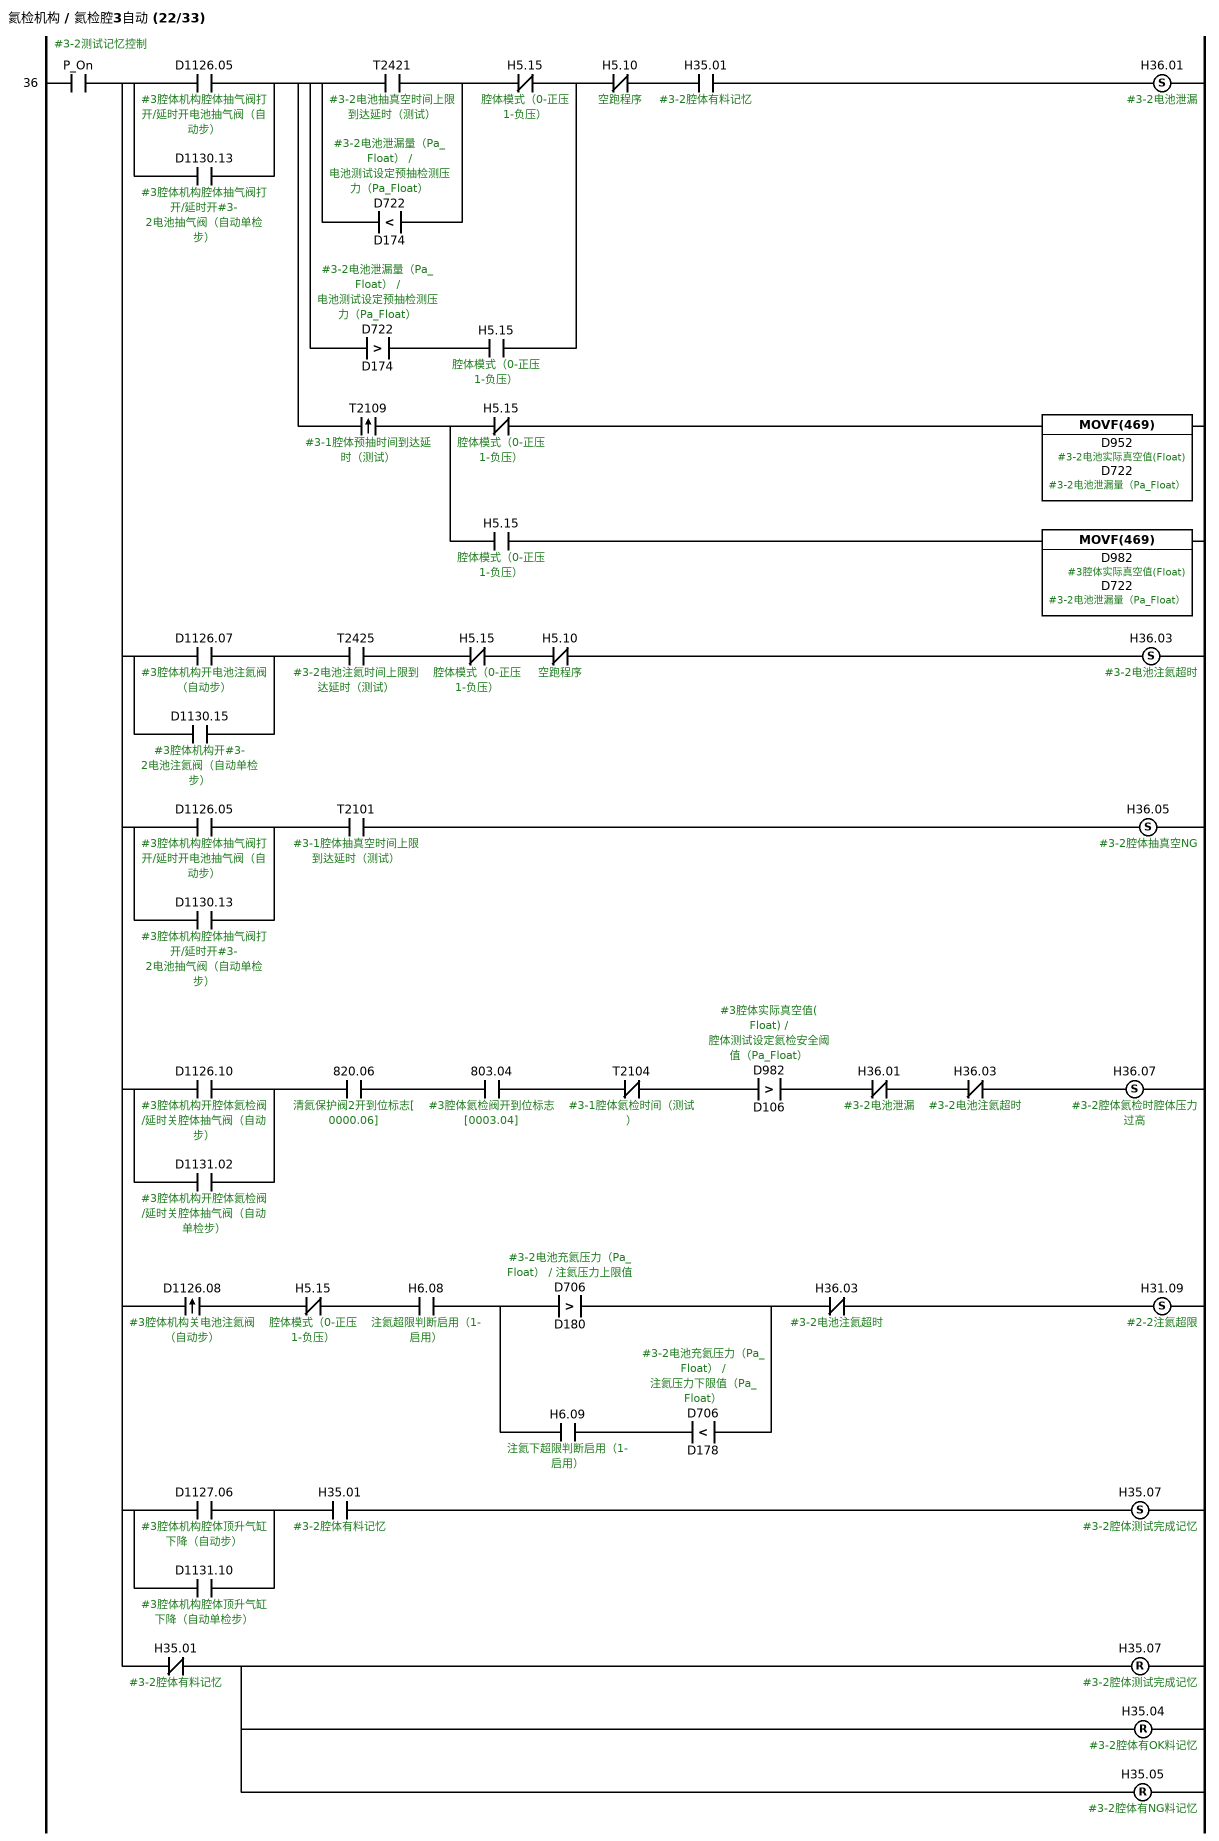
; rung 36: #3-2测试记忆控制
LD P_On
OUT TR0
LD D1126.05  ; #3腔体机构腔体抽气阀打开/延时开电池抽气阀（自动步）
OR D1130.13  ; #3腔体机构腔体抽气阀打开/延时开#3-2电池抽气阀（自动单检步）
ANDLD
OUT TR1
LD T2421  ; #3-2电池抽真空时间上限到达延时（测试）
OR<F(331) D722 D174  ; #3-2电池泄漏量（Pa_Float）, 电池测试设定预抽检测压力（Pa_Float）
ANDNOT H5.15  ; 腔体模式（0-正压 1-负压）
LD>F(333) D722 D174  ; #3-2电池泄漏量（Pa_Float）, 电池测试设定预抽检测压力（Pa_Float）
AND H5.15  ; 腔体模式（0-正压 1-负压）
ORLD
ANDLD
ANDNOT H5.10  ; 空跑程序
AND H35.01  ; #3-2腔体有料记忆
SET H36.01  ; #3-2电池泄漏
LD TR1
@AND T2109  ; #3-1腔体预抽时间到达延时（测试）
OUT TR1
ANDNOT H5.15  ; 腔体模式（0-正压 1-负压）
MOVF(469) D952 D722  ; #3-2电池实际真空值(Float), #3-2电池泄漏量（Pa_Float）
LD TR1
AND H5.15  ; 腔体模式（0-正压 1-负压）
MOVF(469) D982 D722  ; #3腔体实际真空值(Float), #3-2电池泄漏量（Pa_Float）
LD TR0
LD D1126.07  ; #3腔体机构开电池注氦阀（自动步）
OR D1130.15  ; #3腔体机构开#3-2电池注氦阀（自动单检步）
ANDLD
AND T2425  ; #3-2电池注氦时间上限到达延时（测试）
ANDNOT H5.15  ; 腔体模式（0-正压 1-负压）
ANDNOT H5.10  ; 空跑程序
SET H36.03  ; #3-2电池注氦超时
LD TR0
LD D1126.05  ; #3腔体机构腔体抽气阀打开/延时开电池抽气阀（自动步）
OR D1130.13  ; #3腔体机构腔体抽气阀打开/延时开#3-2电池抽气阀（自动单检步）
ANDLD
AND T2101  ; #3-1腔体抽真空时间上限到达延时（测试）
SET H36.05  ; #3-2腔体抽真空NG
LD TR0
LD D1126.10  ; #3腔体机构开腔体氦检阀/延时关腔体抽气阀（自动步）
OR D1131.02  ; #3腔体机构开腔体氦检阀/延时关腔体抽气阀（自动单检步）
ANDLD
AND 820.06  ; 清氦保护阀2开到位标志[0000.06]
AND 803.04  ; #3腔体氦检阀开到位标志[0003.04]
ANDNOT T2104  ; #3-1腔体氦检时间（测试）
AND>F(333) D982 D106  ; #3腔体实际真空值(Float), 腔体测试设定氦检安全阈值（Pa_Float）
ANDNOT H36.01  ; #3-2电池泄漏
ANDNOT H36.03  ; #3-2电池注氦超时
SET H36.07  ; #3-2腔体氦检时腔体压力过高
LD TR0
@AND D1126.08  ; #3腔体机构关电池注氦阀（自动步）
ANDNOT H5.15  ; 腔体模式（0-正压 1-负压）
AND H6.08  ; 注氦超限判断启用（1-启用）
LD>F(333) D706 D180  ; #3-2电池充氦压力（Pa_Float）, 注氦压力上限值
LD H6.09  ; 注氦下超限判断启用（1-启用）
AND<F(331) D706 D178  ; #3-2电池充氦压力（Pa_Float）, 注氦压力下限值（Pa_Float）
ORLD
ANDLD
ANDNOT H36.03  ; #3-2电池注氦超时
SET H31.09  ; #2-2注氦超限
LD TR0
LD D1127.06  ; #3腔体机构腔体顶升气缸下降（自动步）
OR D1131.10  ; #3腔体机构腔体顶升气缸下降（自动单检步）
ANDLD
AND H35.01  ; #3-2腔体有料记忆
SET H35.07  ; #3-2腔体测试完成记忆
LD TR0
ANDNOT H35.01  ; #3-2腔体有料记忆
RSET H35.07  ; #3-2腔体测试完成记忆
RSET H35.04  ; #3-2腔体有OK料记忆
RSET H35.05  ; #3-2腔体有NG料记忆

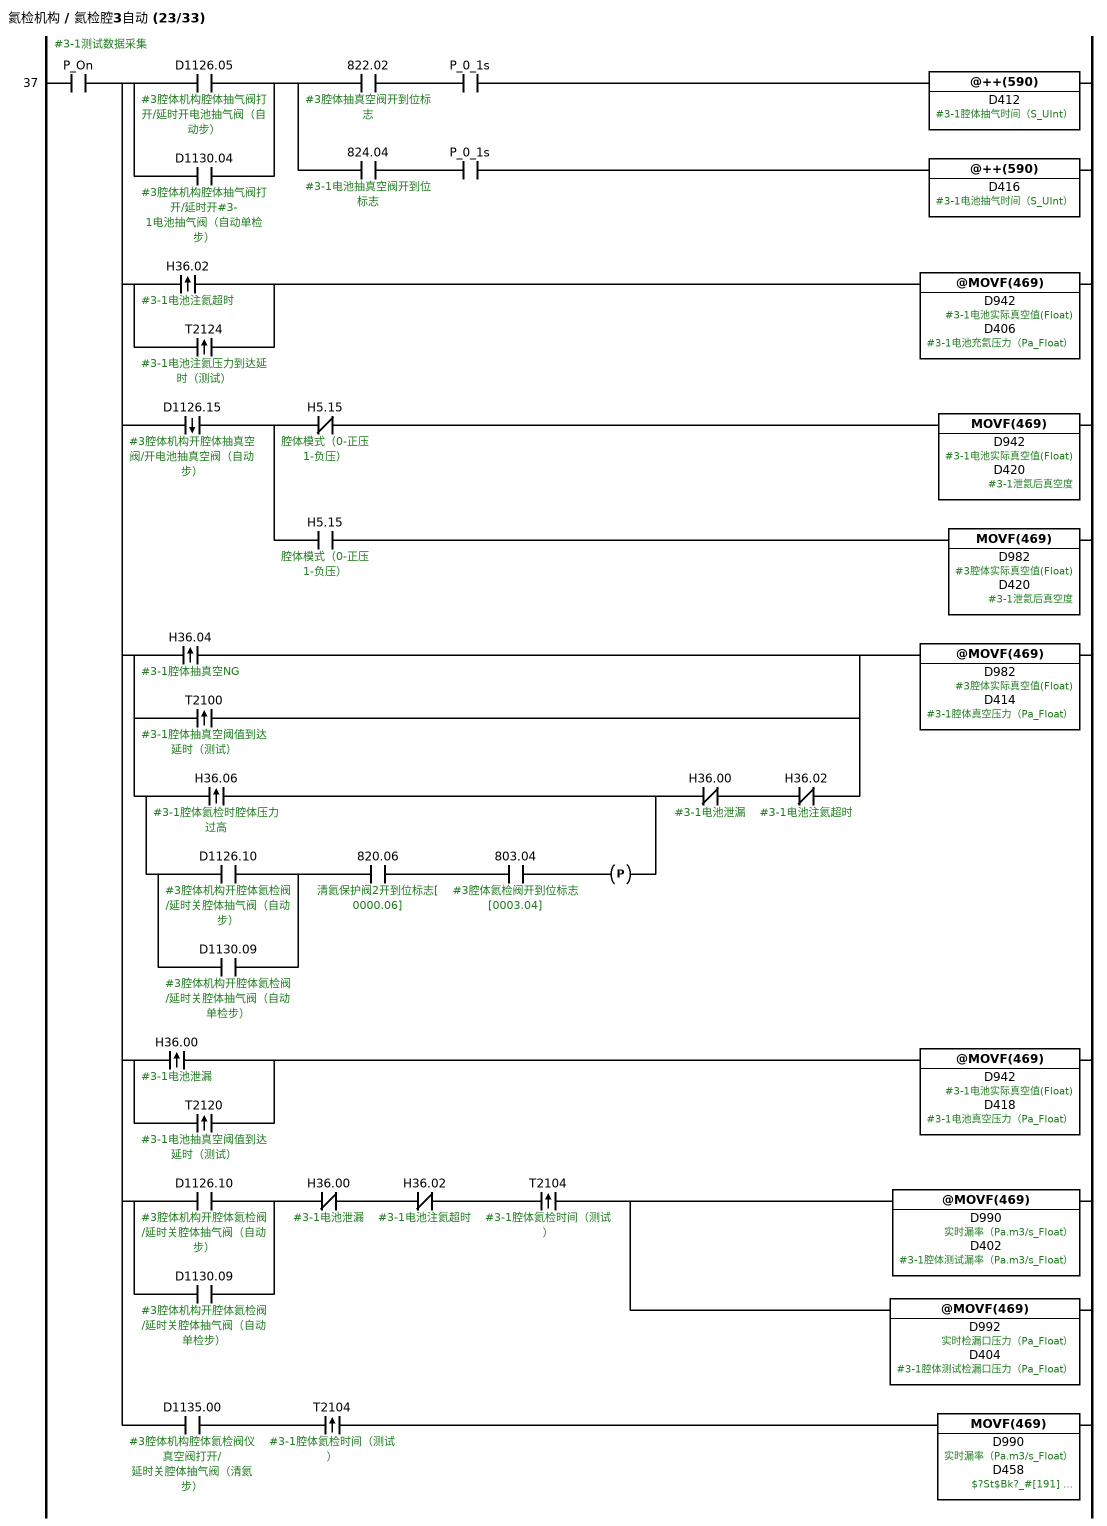
; rung 37: #3-1测试数据采集
LD P_On
OUT TR0
LD D1126.05  ; #3腔体机构腔体抽气阀打开/延时开电池抽气阀（自动步）
OR D1130.04  ; #3腔体机构腔体抽气阀打开/延时开#3-1电池抽气阀（自动单检步）
ANDLD
OUT TR1
AND 822.02  ; #3腔体抽真空阀开到位标志
AND P_0_1s
@++(590) D412  ; #3-1腔体抽气时间（S_UInt）
LD TR1
AND 824.04  ; #3-1电池抽真空阀开到位标志
AND P_0_1s
@++(590) D416  ; #3-1电池抽气时间（S_UInt）
LD TR0
@LD H36.02  ; #3-1电池注氦超时
@OR T2124  ; #3-1电池注氦压力到达延时（测试）
ANDLD
@MOVF(469) D942 D406  ; #3-1电池实际真空值(Float), #3-1电池充氦压力（Pa_Float）
LD TR0
%AND D1126.15  ; #3腔体机构开腔体抽真空阀/开电池抽真空阀（自动步）
OUT TR1
ANDNOT H5.15  ; 腔体模式（0-正压 1-负压）
MOVF(469) D942 D420  ; #3-1电池实际真空值(Float), #3-1泄氦后真空度
LD TR1
AND H5.15  ; 腔体模式（0-正压 1-负压）
MOVF(469) D982 D420  ; #3腔体实际真空值(Float), #3-1泄氦后真空度
LD TR0
@LD H36.04  ; #3-1腔体抽真空NG
@OR T2100  ; #3-1腔体抽真空阈值到达延时（测试）
@LD H36.06  ; #3-1腔体氦检时腔体压力过高
LD D1126.10  ; #3腔体机构开腔体氦检阀/延时关腔体抽气阀（自动步）
OR D1130.09  ; #3腔体机构开腔体氦检阀/延时关腔体抽气阀（自动单检步）
AND 820.06  ; 清氦保护阀2开到位标志[0000.06]
AND 803.04  ; #3腔体氦检阀开到位标志[0003.04]
UP(521)
ORLD
ANDNOT H36.00  ; #3-1电池泄漏
ANDNOT H36.02  ; #3-1电池注氦超时
ORLD
ANDLD
@MOVF(469) D982 D414  ; #3腔体实际真空值(Float), #3-1腔体真空压力（Pa_Float）
LD TR0
@LD H36.00  ; #3-1电池泄漏
@OR T2120  ; #3-1电池抽真空阈值到达延时（测试）
ANDLD
@MOVF(469) D942 D418  ; #3-1电池实际真空值(Float), #3-1电池真空压力（Pa_Float）
LD TR0
LD D1126.10  ; #3腔体机构开腔体氦检阀/延时关腔体抽气阀（自动步）
OR D1130.09  ; #3腔体机构开腔体氦检阀/延时关腔体抽气阀（自动单检步）
ANDLD
ANDNOT H36.00  ; #3-1电池泄漏
ANDNOT H36.02  ; #3-1电池注氦超时
@AND T2104  ; #3-1腔体氦检时间（测试）
@MOVF(469) D990 D402  ; 实时漏率（Pa.m3/s_Float）, #3-1腔体测试漏率（Pa.m3/s_Float）
@MOVF(469) D992 D404  ; 实时检漏口压力（Pa_Float）, #3-1腔体测试检漏口压力（Pa_Float）
LD TR0
AND D1135.00  ; #3腔体机构腔体氦检阀仪真空阀打开/延时关腔体抽气阀（清氦步）
@AND T2104  ; #3-1腔体氦检时间（测试）
MOVF(469) D990 D458  ; 实时漏率（Pa.m3/s_Float）, $?St$Bk?_#[191] / #3-1清氦泄漏率（清氦） / $?St$Bk?_#[191]

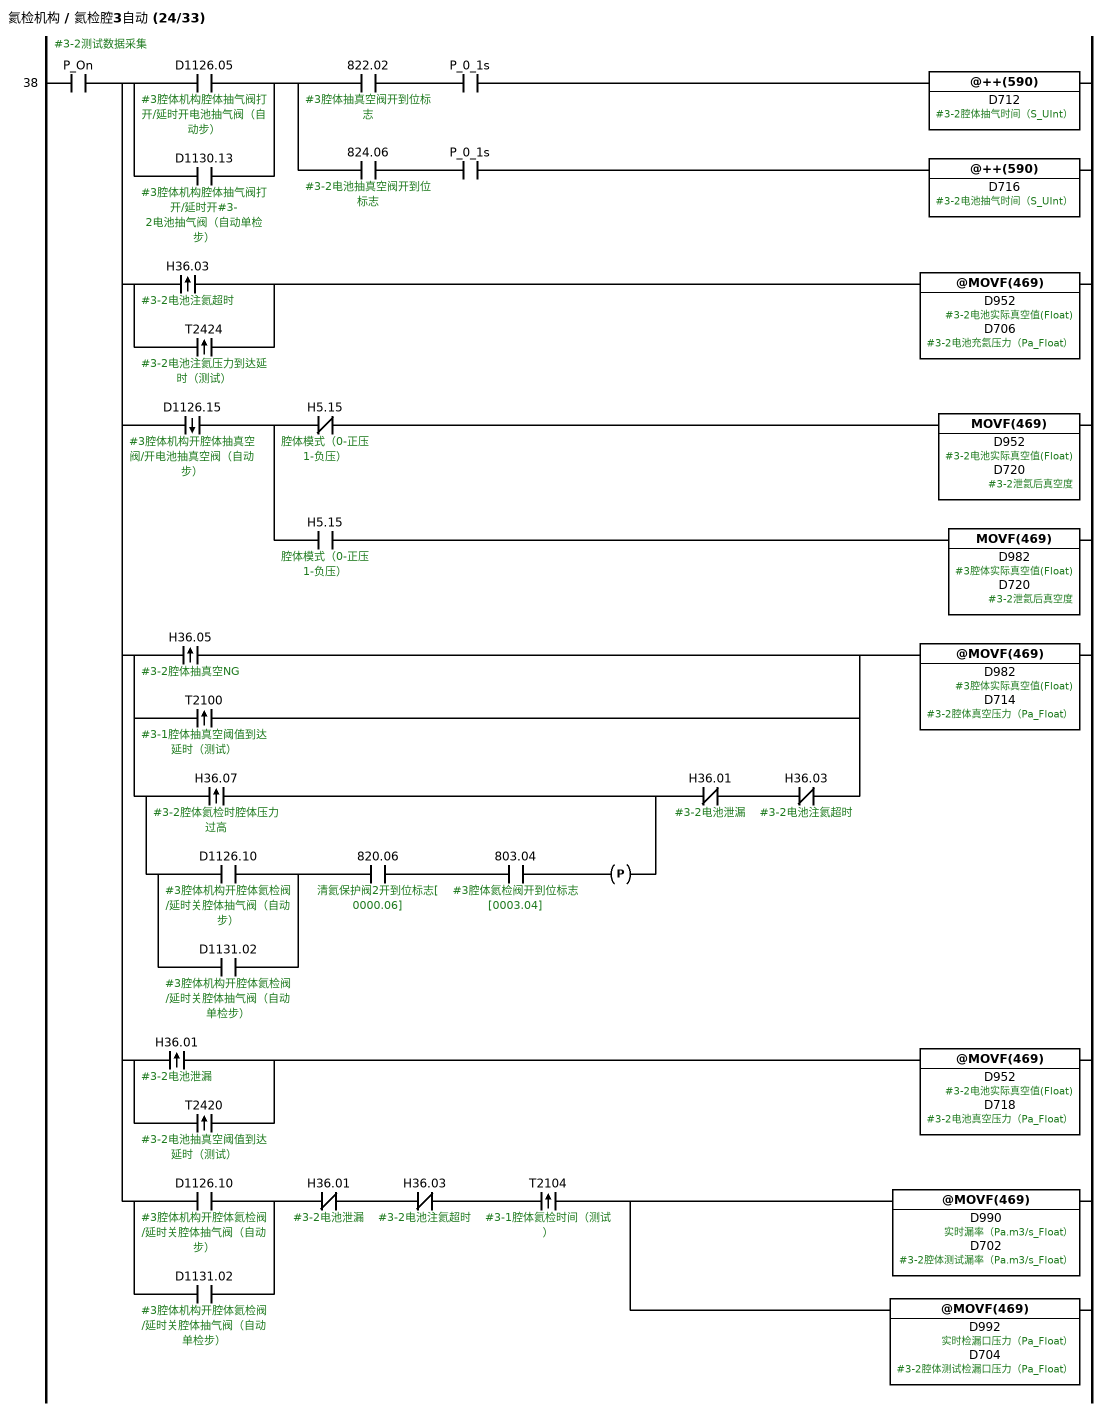
; rung 38: #3-2测试数据采集
LD P_On
OUT TR0
LD D1126.05  ; #3腔体机构腔体抽气阀打开/延时开电池抽气阀（自动步）
OR D1130.13  ; #3腔体机构腔体抽气阀打开/延时开#3-2电池抽气阀（自动单检步）
ANDLD
OUT TR1
AND 822.02  ; #3腔体抽真空阀开到位标志
AND P_0_1s
@++(590) D712  ; #3-2腔体抽气时间（S_UInt）
LD TR1
AND 824.06  ; #3-2电池抽真空阀开到位标志
AND P_0_1s
@++(590) D716  ; #3-2电池抽气时间（S_UInt）
LD TR0
@LD H36.03  ; #3-2电池注氦超时
@OR T2424  ; #3-2电池注氦压力到达延时（测试）
ANDLD
@MOVF(469) D952 D706  ; #3-2电池实际真空值(Float), #3-2电池充氦压力（Pa_Float）
LD TR0
%AND D1126.15  ; #3腔体机构开腔体抽真空阀/开电池抽真空阀（自动步）
OUT TR1
ANDNOT H5.15  ; 腔体模式（0-正压 1-负压）
MOVF(469) D952 D720  ; #3-2电池实际真空值(Float), #3-2泄氦后真空度
LD TR1
AND H5.15  ; 腔体模式（0-正压 1-负压）
MOVF(469) D982 D720  ; #3腔体实际真空值(Float), #3-2泄氦后真空度
LD TR0
@LD H36.05  ; #3-2腔体抽真空NG
@OR T2100  ; #3-1腔体抽真空阈值到达延时（测试）
@LD H36.07  ; #3-2腔体氦检时腔体压力过高
LD D1126.10  ; #3腔体机构开腔体氦检阀/延时关腔体抽气阀（自动步）
OR D1131.02  ; #3腔体机构开腔体氦检阀/延时关腔体抽气阀（自动单检步）
AND 820.06  ; 清氦保护阀2开到位标志[0000.06]
AND 803.04  ; #3腔体氦检阀开到位标志[0003.04]
UP(521)
ORLD
ANDNOT H36.01  ; #3-2电池泄漏
ANDNOT H36.03  ; #3-2电池注氦超时
ORLD
ANDLD
@MOVF(469) D982 D714  ; #3腔体实际真空值(Float), #3-2腔体真空压力（Pa_Float）
LD TR0
@LD H36.01  ; #3-2电池泄漏
@OR T2420  ; #3-2电池抽真空阈值到达延时（测试）
ANDLD
@MOVF(469) D952 D718  ; #3-2电池实际真空值(Float), #3-2电池真空压力（Pa_Float）
LD TR0
LD D1126.10  ; #3腔体机构开腔体氦检阀/延时关腔体抽气阀（自动步）
OR D1131.02  ; #3腔体机构开腔体氦检阀/延时关腔体抽气阀（自动单检步）
ANDLD
ANDNOT H36.01  ; #3-2电池泄漏
ANDNOT H36.03  ; #3-2电池注氦超时
@AND T2104  ; #3-1腔体氦检时间（测试）
@MOVF(469) D990 D702  ; 实时漏率（Pa.m3/s_Float）, #3-2腔体测试漏率（Pa.m3/s_Float）
@MOVF(469) D992 D704  ; 实时检漏口压力（Pa_Float）, #3-2腔体测试检漏口压力（Pa_Float）

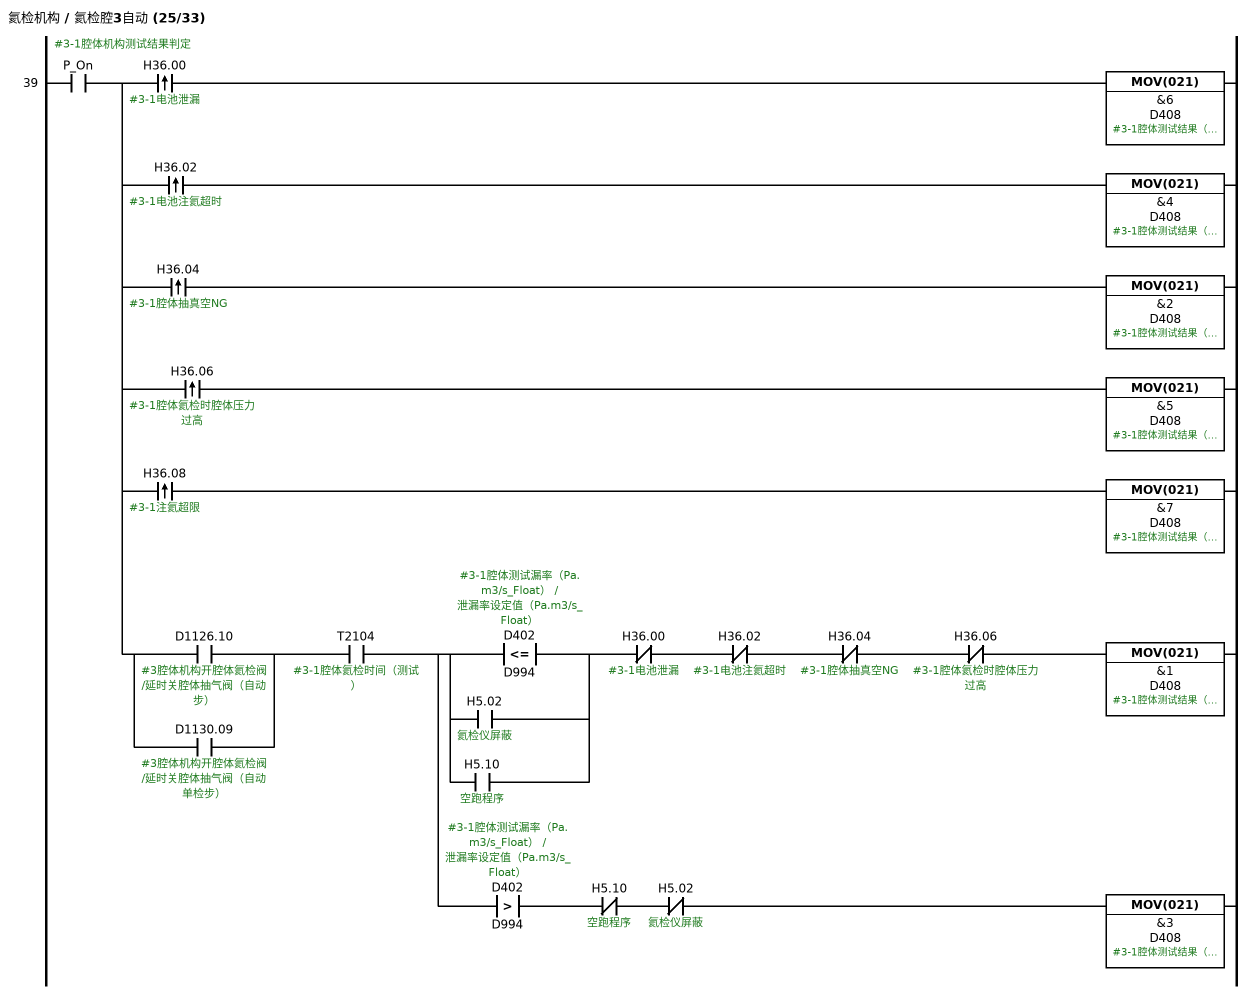
; rung 39: #3-1腔体机构测试结果判定
LD P_On
OUT TR0
@AND H36.00  ; #3-1电池泄漏
MOV(021) &6 D408  ; #3-1腔体测试结果（1 OK，2腔体泄漏，3气密NG，4注氦超时，5氦检异常，6电池泄漏，7注氦NG，8氦嘴泄漏）
LD TR0
@AND H36.02  ; #3-1电池注氦超时
MOV(021) &4 D408  ; #3-1腔体测试结果（1 OK，2腔体泄漏，3气密NG，4注氦超时，5氦检异常，6电池泄漏，7注氦NG，8氦嘴泄漏）
LD TR0
@AND H36.04  ; #3-1腔体抽真空NG
MOV(021) &2 D408  ; #3-1腔体测试结果（1 OK，2腔体泄漏，3气密NG，4注氦超时，5氦检异常，6电池泄漏，7注氦NG，8氦嘴泄漏）
LD TR0
@AND H36.06  ; #3-1腔体氦检时腔体压力过高
MOV(021) &5 D408  ; #3-1腔体测试结果（1 OK，2腔体泄漏，3气密NG，4注氦超时，5氦检异常，6电池泄漏，7注氦NG，8氦嘴泄漏）
LD TR0
@AND H36.08  ; #3-1注氦超限
MOV(021) &7 D408  ; #3-1腔体测试结果（1 OK，2腔体泄漏，3气密NG，4注氦超时，5氦检异常，6电池泄漏，7注氦NG，8氦嘴泄漏）
LD TR0
LD D1126.10  ; #3腔体机构开腔体氦检阀/延时关腔体抽气阀（自动步）
OR D1130.09  ; #3腔体机构开腔体氦检阀/延时关腔体抽气阀（自动单检步）
ANDLD
AND T2104  ; #3-1腔体氦检时间（测试）
OUT TR0
LD<=F(332) D402 D994  ; #3-1腔体测试漏率（Pa.m3/s_Float）, 泄漏率设定值（Pa.m3/s_Float）
OR H5.02  ; 氦检仪屏蔽
OR H5.10  ; 空跑程序
ANDLD
ANDNOT H36.00  ; #3-1电池泄漏
ANDNOT H36.02  ; #3-1电池注氦超时
ANDNOT H36.04  ; #3-1腔体抽真空NG
ANDNOT H36.06  ; #3-1腔体氦检时腔体压力过高
MOV(021) &1 D408  ; #3-1腔体测试结果（1 OK，2腔体泄漏，3气密NG，4注氦超时，5氦检异常，6电池泄漏，7注氦NG，8氦嘴泄漏）
LD TR0
AND>F(333) D402 D994  ; #3-1腔体测试漏率（Pa.m3/s_Float）, 泄漏率设定值（Pa.m3/s_Float）
ANDNOT H5.10  ; 空跑程序
ANDNOT H5.02  ; 氦检仪屏蔽
MOV(021) &3 D408  ; #3-1腔体测试结果（1 OK，2腔体泄漏，3气密NG，4注氦超时，5氦检异常，6电池泄漏，7注氦NG，8氦嘴泄漏）

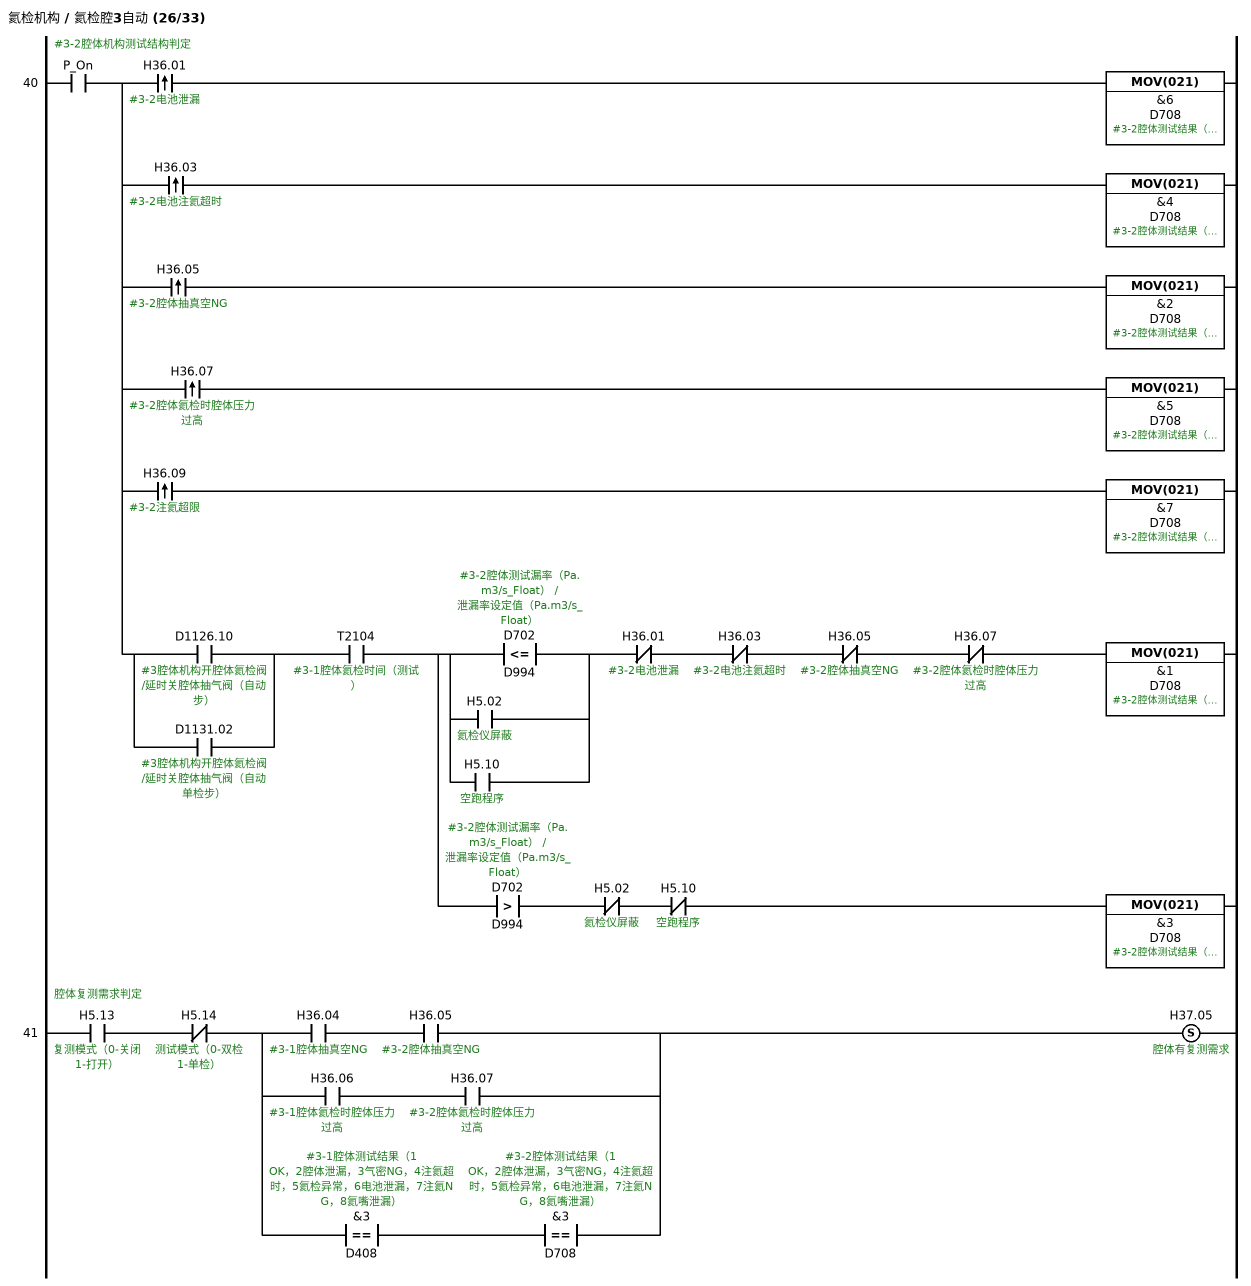
; rung 40: #3-2腔体机构测试结构判定
LD P_On
OUT TR0
@AND H36.01  ; #3-2电池泄漏
MOV(021) &6 D708  ; #3-2腔体测试结果（1 OK，2腔体泄漏，3气密NG，4注氦超时，5氦检异常，6电池泄漏，7注氦NG，8氦嘴泄漏）
LD TR0
@AND H36.03  ; #3-2电池注氦超时
MOV(021) &4 D708  ; #3-2腔体测试结果（1 OK，2腔体泄漏，3气密NG，4注氦超时，5氦检异常，6电池泄漏，7注氦NG，8氦嘴泄漏）
LD TR0
@AND H36.05  ; #3-2腔体抽真空NG
MOV(021) &2 D708  ; #3-2腔体测试结果（1 OK，2腔体泄漏，3气密NG，4注氦超时，5氦检异常，6电池泄漏，7注氦NG，8氦嘴泄漏）
LD TR0
@AND H36.07  ; #3-2腔体氦检时腔体压力过高
MOV(021) &5 D708  ; #3-2腔体测试结果（1 OK，2腔体泄漏，3气密NG，4注氦超时，5氦检异常，6电池泄漏，7注氦NG，8氦嘴泄漏）
LD TR0
@AND H36.09  ; #3-2注氦超限
MOV(021) &7 D708  ; #3-2腔体测试结果（1 OK，2腔体泄漏，3气密NG，4注氦超时，5氦检异常，6电池泄漏，7注氦NG，8氦嘴泄漏）
LD TR0
LD D1126.10  ; #3腔体机构开腔体氦检阀/延时关腔体抽气阀（自动步）
OR D1131.02  ; #3腔体机构开腔体氦检阀/延时关腔体抽气阀（自动单检步）
ANDLD
AND T2104  ; #3-1腔体氦检时间（测试）
OUT TR0
LD<=F(332) D702 D994  ; #3-2腔体测试漏率（Pa.m3/s_Float）, 泄漏率设定值（Pa.m3/s_Float）
OR H5.02  ; 氦检仪屏蔽
OR H5.10  ; 空跑程序
ANDLD
ANDNOT H36.01  ; #3-2电池泄漏
ANDNOT H36.03  ; #3-2电池注氦超时
ANDNOT H36.05  ; #3-2腔体抽真空NG
ANDNOT H36.07  ; #3-2腔体氦检时腔体压力过高
MOV(021) &1 D708  ; #3-2腔体测试结果（1 OK，2腔体泄漏，3气密NG，4注氦超时，5氦检异常，6电池泄漏，7注氦NG，8氦嘴泄漏）
LD TR0
AND>F(333) D702 D994  ; #3-2腔体测试漏率（Pa.m3/s_Float）, 泄漏率设定值（Pa.m3/s_Float）
ANDNOT H5.02  ; 氦检仪屏蔽
ANDNOT H5.10  ; 空跑程序
MOV(021) &3 D708  ; #3-2腔体测试结果（1 OK，2腔体泄漏，3气密NG，4注氦超时，5氦检异常，6电池泄漏，7注氦NG，8氦嘴泄漏）
; rung 41: 腔体复测需求判定
LD H5.13  ; 复测模式（0-关闭 1-打开）
ANDNOT H5.14  ; 测试模式（0-双检 1-单检）
LD H36.04  ; #3-1腔体抽真空NG
AND H36.05  ; #3-2腔体抽真空NG
LD H36.06  ; #3-1腔体氦检时腔体压力过高
AND H36.07  ; #3-2腔体氦检时腔体压力过高
ORLD
LD=(300) &3 D408  ; #3-1腔体测试结果（1 OK，2腔体泄漏，3气密NG，4注氦超时，5氦检异常，6电池泄漏，7注氦NG，8氦嘴泄漏）
AND=(300) &3 D708  ; #3-2腔体测试结果（1 OK，2腔体泄漏，3气密NG，4注氦超时，5氦检异常，6电池泄漏，7注氦NG，8氦嘴泄漏）
ORLD
ANDLD
SET H37.05  ; 腔体有复测需求

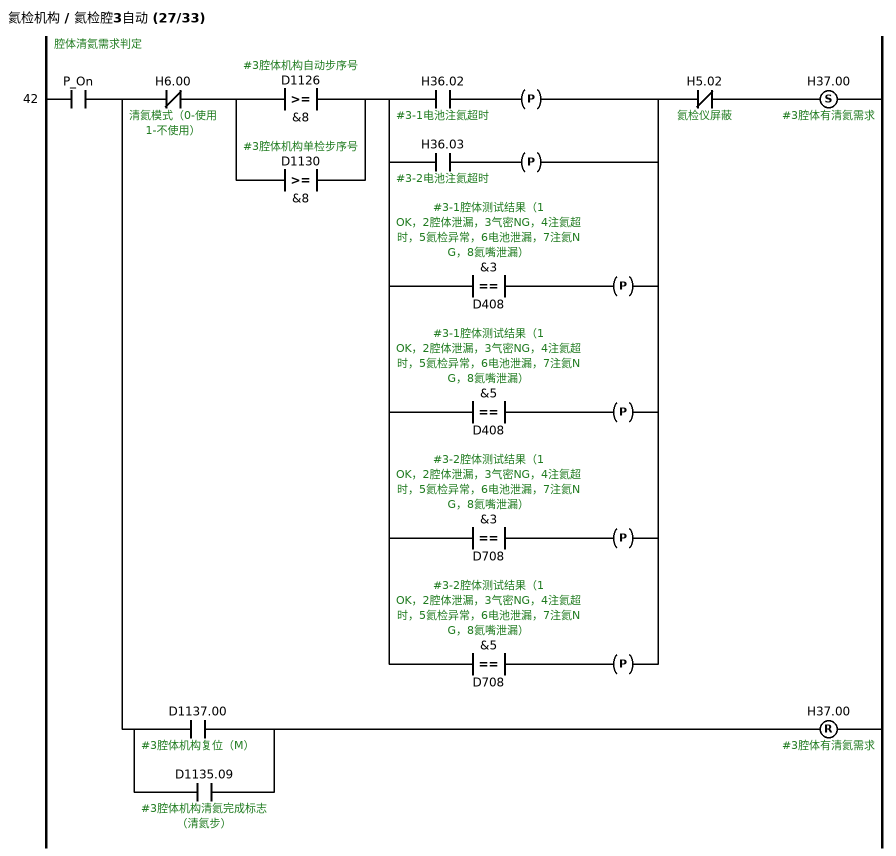
; rung 42: 腔体清氦需求判定
LD P_On
OUT TR0
ANDNOT H6.00  ; 清氦模式（0-使用 1-不使用）
LD>=L(326) D1126 &8  ; #3腔体机构自动步序号
OR>=L(326) D1130 &8  ; #3腔体机构单检步序号
ANDLD
LD H36.02  ; #3-1电池注氦超时
UP(521)
LD H36.03  ; #3-2电池注氦超时
UP(521)
ORLD
LD=(300) &3 D408  ; #3-1腔体测试结果（1 OK，2腔体泄漏，3气密NG，4注氦超时，5氦检异常，6电池泄漏，7注氦NG，8氦嘴泄漏）
UP(521)
ORLD
LD=(300) &5 D408  ; #3-1腔体测试结果（1 OK，2腔体泄漏，3气密NG，4注氦超时，5氦检异常，6电池泄漏，7注氦NG，8氦嘴泄漏）
UP(521)
ORLD
LD=(300) &3 D708  ; #3-2腔体测试结果（1 OK，2腔体泄漏，3气密NG，4注氦超时，5氦检异常，6电池泄漏，7注氦NG，8氦嘴泄漏）
UP(521)
ORLD
LD=(300) &5 D708  ; #3-2腔体测试结果（1 OK，2腔体泄漏，3气密NG，4注氦超时，5氦检异常，6电池泄漏，7注氦NG，8氦嘴泄漏）
UP(521)
ORLD
ANDLD
ANDNOT H5.02  ; 氦检仪屏蔽
SET H37.00  ; #3腔体有清氦需求
LD TR0
LD D1137.00  ; #3腔体机构复位（M）
OR D1135.09  ; #3腔体机构清氦完成标志（清氦步）
ANDLD
RSET H37.00  ; #3腔体有清氦需求

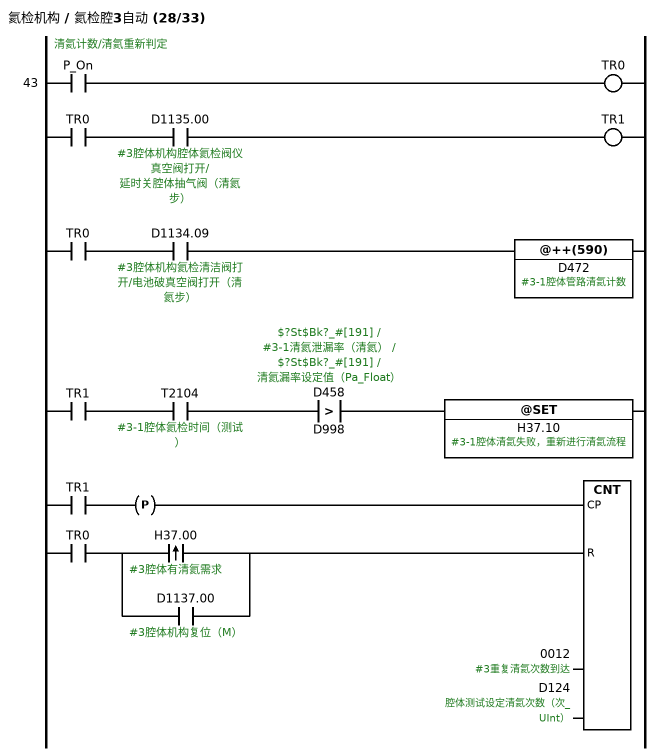
; rung 43: 清氦计数/清氦重新判定
LD P_On
OUT TR0
AND D1134.09  ; #3腔体机构氦检清洁阀打开/电池破真空阀打开（清氦步）
@++(590) D472  ; #3-1腔体管路清氦计数
LD TR0
AND D1135.00  ; #3腔体机构腔体氦检阀仪真空阀打开/延时关腔体抽气阀（清氦步）
OUT TR1
AND T2104  ; #3-1腔体氦检时间（测试）
AND>F(333) D458 D998  ; $?St$Bk?_#[191] / #3-1清氦泄漏率（清氦） / $?St$Bk?_#[191], 清氦漏率设定值（Pa_Float）
@SET H37.10  ; #3-1腔体清氦失败，重新进行清氦流程
LD TR1
UP(521)
LD TR0
@LD H37.00  ; #3腔体有清氦需求
OR D1137.00  ; #3腔体机构复位（M）
ANDLD
CNT 0012 D124  ; 腔体测试设定清氦次数（次_UInt）, #3重复清氦次数到达

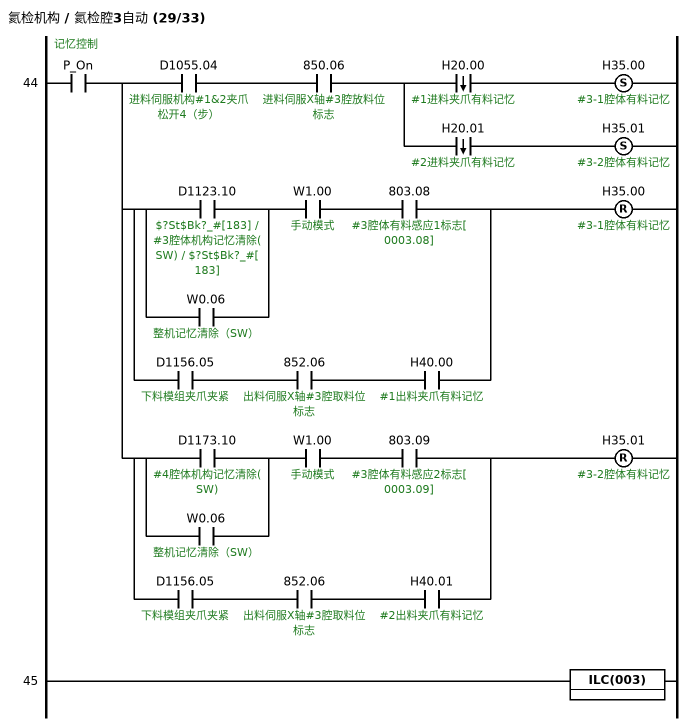
; rung 44: 记忆控制
LD P_On
OUT TR0
AND D1055.04  ; 进料伺服机构#1&2夹爪松开4（步）
AND 850.06  ; 进料伺服X轴#3腔放料位标志
OUT TR1
%AND H20.00  ; #1进料夹爪有料记忆
SET H35.00  ; #3-1腔体有料记忆
LD TR1
%AND H20.01  ; #2进料夹爪有料记忆
SET H35.01  ; #3-2腔体有料记忆
LD TR0
LD D1123.10  ; $?St$Bk?_#[183] / #3腔体机构记忆清除(SW) / $?St$Bk?_#[183]
OR W0.06  ; 整机记忆清除（SW）
AND W1.00  ; 手动模式
AND 803.08  ; #3腔体有料感应1标志[0003.08]
LD D1156.05  ; 下料模组夹爪夹紧
AND 852.06  ; 出料伺服X轴#3腔取料位标志
AND H40.00  ; #1出料夹爪有料记忆
ORLD
ANDLD
RSET H35.00  ; #3-1腔体有料记忆
LD TR0
LD D1173.10  ; #4腔体机构记忆清除(SW)
OR W0.06  ; 整机记忆清除（SW）
AND W1.00  ; 手动模式
AND 803.09  ; #3腔体有料感应2标志[0003.09]
LD D1156.05  ; 下料模组夹爪夹紧
AND 852.06  ; 出料伺服X轴#3腔取料位标志
AND H40.01  ; #2出料夹爪有料记忆
ORLD
ANDLD
RSET H35.01  ; #3-2腔体有料记忆
; rung 45
ILC(003)

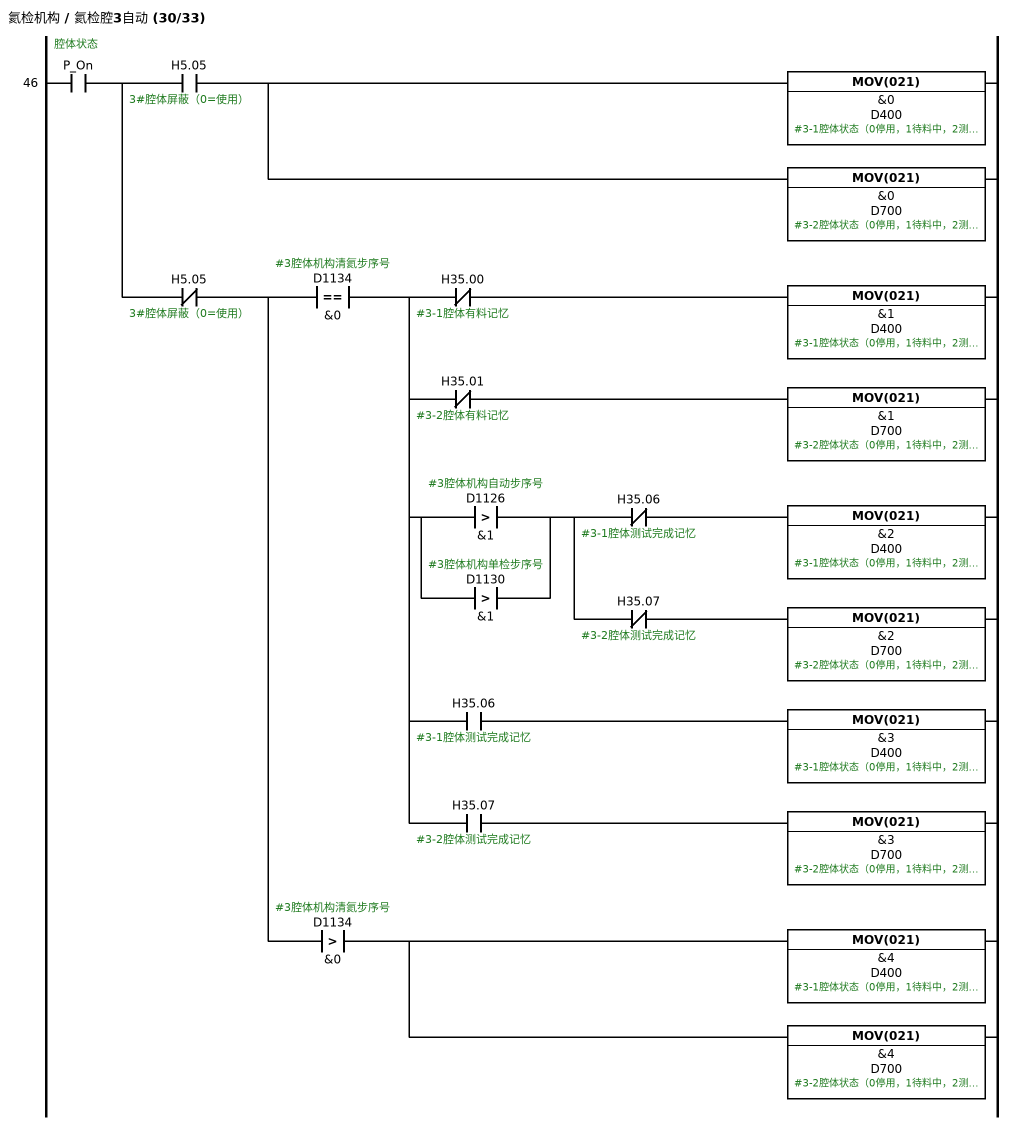
; rung 46: 腔体状态
LD P_On
OUT TR0
AND H5.05  ; 3#腔体屏蔽（0=使用）
MOV(021) &0 D400  ; #3-1腔体状态（0停用，1待料中，2测试中，3测试完成，4-清氦中）
MOV(021) &0 D700  ; #3-2腔体状态（0停用，1待料中，2测试中，3测试完成，4-清氦中）
LD TR0
ANDNOT H5.05  ; 3#腔体屏蔽（0=使用）
OUT TR0
AND=L(301) D1134 &0  ; #3腔体机构清氦步序号
OUT TR1
ANDNOT H35.00  ; #3-1腔体有料记忆
MOV(021) &1 D400  ; #3-1腔体状态（0停用，1待料中，2测试中，3测试完成，4-清氦中）
LD TR1
ANDNOT H35.01  ; #3-2腔体有料记忆
MOV(021) &1 D700  ; #3-2腔体状态（0停用，1待料中，2测试中，3测试完成，4-清氦中）
LD TR1
LD>L(321) D1126 &1  ; #3腔体机构自动步序号
OR>L(321) D1130 &1  ; #3腔体机构单检步序号
ANDLD
OUT TR2
ANDNOT H35.06  ; #3-1腔体测试完成记忆
MOV(021) &2 D400  ; #3-1腔体状态（0停用，1待料中，2测试中，3测试完成，4-清氦中）
LD TR2
ANDNOT H35.07  ; #3-2腔体测试完成记忆
MOV(021) &2 D700  ; #3-2腔体状态（0停用，1待料中，2测试中，3测试完成，4-清氦中）
LD TR1
AND H35.06  ; #3-1腔体测试完成记忆
MOV(021) &3 D400  ; #3-1腔体状态（0停用，1待料中，2测试中，3测试完成，4-清氦中）
LD TR1
AND H35.07  ; #3-2腔体测试完成记忆
MOV(021) &3 D700  ; #3-2腔体状态（0停用，1待料中，2测试中，3测试完成，4-清氦中）
LD TR0
AND>L(321) D1134 &0  ; #3腔体机构清氦步序号
MOV(021) &4 D400  ; #3-1腔体状态（0停用，1待料中，2测试中，3测试完成，4-清氦中）
MOV(021) &4 D700  ; #3-2腔体状态（0停用，1待料中，2测试中，3测试完成，4-清氦中）

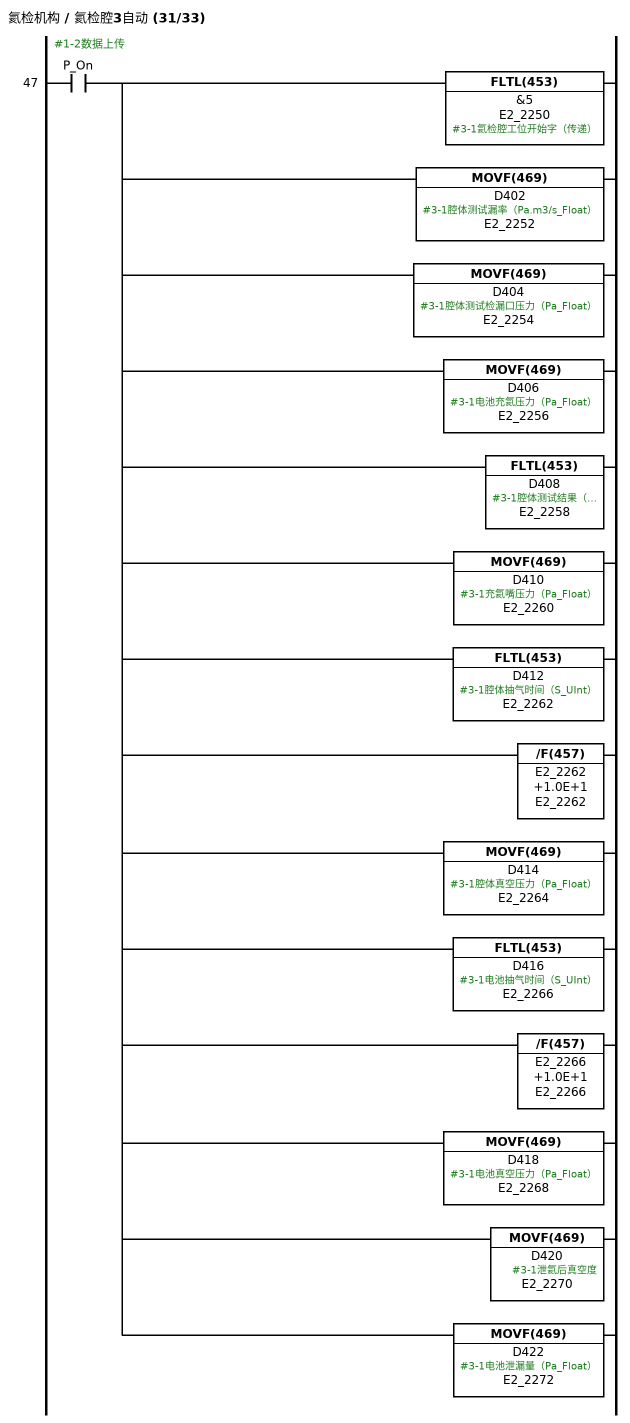
; rung 47: #1-2数据上传
LD P_On
FLTL(453) &5 E2_2250  ; #3-1氦检腔工位开始字（传递）
MOVF(469) D402 E2_2252  ; #3-1腔体测试漏率（Pa.m3/s_Float）
MOVF(469) D404 E2_2254  ; #3-1腔体测试检漏口压力（Pa_Float）
MOVF(469) D406 E2_2256  ; #3-1电池充氦压力（Pa_Float）
FLTL(453) D408 E2_2258  ; #3-1腔体测试结果（1 OK，2腔体泄漏，3气密NG，4注氦超时，5氦检异常，6电池泄漏，7注氦NG，8氦嘴泄漏）
MOVF(469) D410 E2_2260  ; #3-1充氦嘴压力（Pa_Float）
FLTL(453) D412 E2_2262  ; #3-1腔体抽气时间（S_UInt）
/F(457) E2_2262 +1.0E+1 E2_2262
MOVF(469) D414 E2_2264  ; #3-1腔体真空压力（Pa_Float）
FLTL(453) D416 E2_2266  ; #3-1电池抽气时间（S_UInt）
/F(457) E2_2266 +1.0E+1 E2_2266
MOVF(469) D418 E2_2268  ; #3-1电池真空压力（Pa_Float）
MOVF(469) D420 E2_2270  ; #3-1泄氦后真空度
MOVF(469) D422 E2_2272  ; #3-1电池泄漏量（Pa_Float）

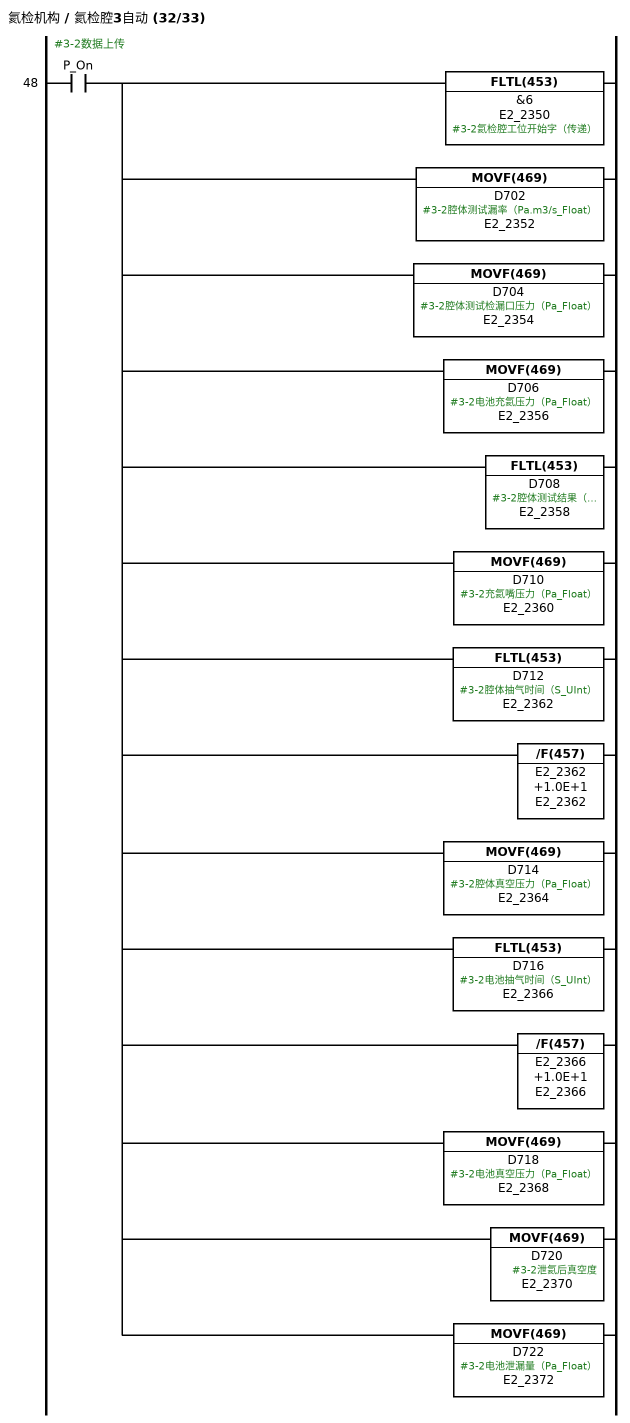
; rung 48: #3-2数据上传
LD P_On
FLTL(453) &6 E2_2350  ; #3-2氦检腔工位开始字（传递）
MOVF(469) D702 E2_2352  ; #3-2腔体测试漏率（Pa.m3/s_Float）
MOVF(469) D704 E2_2354  ; #3-2腔体测试检漏口压力（Pa_Float）
MOVF(469) D706 E2_2356  ; #3-2电池充氦压力（Pa_Float）
FLTL(453) D708 E2_2358  ; #3-2腔体测试结果（1 OK，2腔体泄漏，3气密NG，4注氦超时，5氦检异常，6电池泄漏，7注氦NG，8氦嘴泄漏）
MOVF(469) D710 E2_2360  ; #3-2充氦嘴压力（Pa_Float）
FLTL(453) D712 E2_2362  ; #3-2腔体抽气时间（S_UInt）
/F(457) E2_2362 +1.0E+1 E2_2362
MOVF(469) D714 E2_2364  ; #3-2腔体真空压力（Pa_Float）
FLTL(453) D716 E2_2366  ; #3-2电池抽气时间（S_UInt）
/F(457) E2_2366 +1.0E+1 E2_2366
MOVF(469) D718 E2_2368  ; #3-2电池真空压力（Pa_Float）
MOVF(469) D720 E2_2370  ; #3-2泄氦后真空度
MOVF(469) D722 E2_2372  ; #3-2电池泄漏量（Pa_Float）

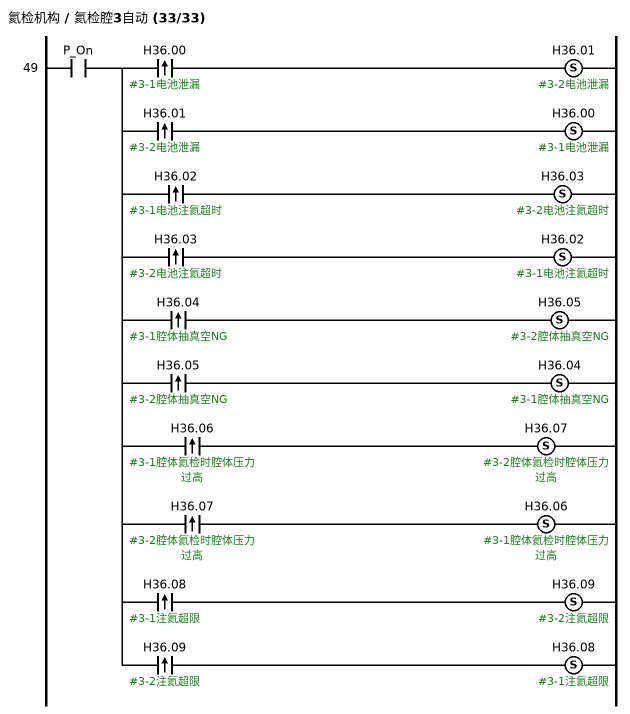
; rung 49
LD P_On
OUT TR0
@AND H36.00  ; #3-1电池泄漏
SET H36.01  ; #3-2电池泄漏
LD TR0
@AND H36.01  ; #3-2电池泄漏
SET H36.00  ; #3-1电池泄漏
LD TR0
@AND H36.02  ; #3-1电池注氦超时
SET H36.03  ; #3-2电池注氦超时
LD TR0
@AND H36.03  ; #3-2电池注氦超时
SET H36.02  ; #3-1电池注氦超时
LD TR0
@AND H36.04  ; #3-1腔体抽真空NG
SET H36.05  ; #3-2腔体抽真空NG
LD TR0
@AND H36.05  ; #3-2腔体抽真空NG
SET H36.04  ; #3-1腔体抽真空NG
LD TR0
@AND H36.06  ; #3-1腔体氦检时腔体压力过高
SET H36.07  ; #3-2腔体氦检时腔体压力过高
LD TR0
@AND H36.07  ; #3-2腔体氦检时腔体压力过高
SET H36.06  ; #3-1腔体氦检时腔体压力过高
LD TR0
@AND H36.08  ; #3-1注氦超限
SET H36.09  ; #3-2注氦超限
LD TR0
@AND H36.09  ; #3-2注氦超限
SET H36.08  ; #3-1注氦超限

### Section 氦检腔4自动

